KUKA KRL program: EPS_2_251455_MH62A_A_20251003045105.src

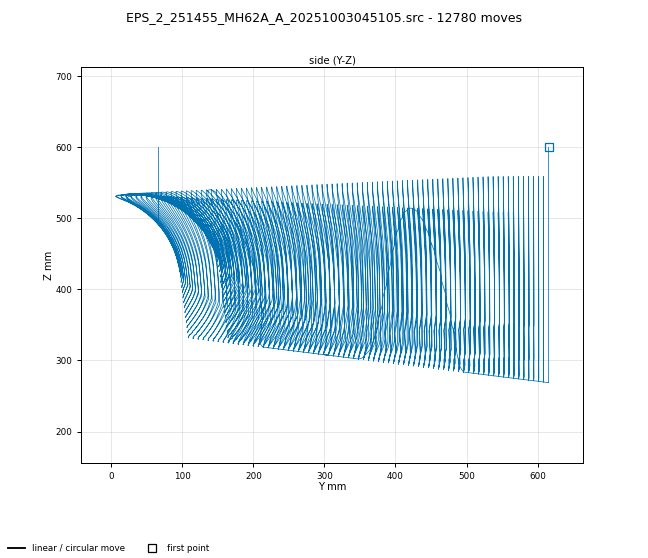
[picture p0: tool path of EPS_2_251455_MH62A_A_20251003045105.src, 12780 of 12782 moves have a stored position in this frame; points joined in program order, loops and branches not executed]
&ACCESS RVP
&REL 4
&COMMENT QRS 19112012
&PARAM EDITMASK = *
DEF PART()
EXT BAS (BAS_COMMAND :IN,REAL :IN )
INT I
BAS (#INITMOV,0 )

;KUKA QRS Post kuka4.cps  Date:22-06-2017 !

File_ID=2872

QRS_PRE_INIT()

;Init var - Until changes are made in qrs_pre_init
Outlet_Square_prg=0
Inlet_1_Square_prg=0
Inlet_2_Square_prg=0
Inlet_3_Square_prg=0
Inlet_4_Square_prg=0
Inlet_5_Square_prg=0

Outlet_1={X 0.000, Y 535.490, Z 458.500, B 0.000, E1 0.000 }
Inlet_1={X 0.000, Y 539.060, Z 408.500, B 0.000, E1 171.000 }
Outlet_1_type=201
Inlet_1_type=201
;QRS#1=Sidecore dimensions
;QRS#2=200-8" PVC SDR 35
;QRS#3=200-8" PVC SDR 35
;QRS#4=
;QRS#5=
;QRS#6=
;QRS#7=
;QRS#8=
;QRS#9=12-08 PSX
;QRS#10=12-08 PSX
;QRS#11=
;QRS#12=
;QRS#13=
;QRS#14=
;QRS#15=
;QRS#16=1220x127x838 2,75'
;QRS#17=EPS Height
;QRS#18=559
;QRS#19=*
;QRS#20= UPDATED VERSION 22-06-2017
;QRS#21=*
Outlet_Square=0100
Inlet_1_Square=0100
Inlet_2_Square=0
Inlet_3_Square=0
Inlet_4_Square=0
Inlet_5_Square=0
Mill_Square=1
Outlet_Square_Prg=204
Inlet_1_Square_prg=204

QRS_INIT()

$ADVANCE=5

; T1
PTP {E1 173.608,E2 173.608}
PTP {X 0,Y 615.498,A -85,B 0,C 180,E1 173.608,E2 173.608,E3 0,E4 0,E5 0,E6 0}
QRS_SPEED_INIT()
LIN {X 0,Y 615.498,Z 600,A -85,B 0,C 180,E1 173.608,E2 173.608,E3 0,E4 0,E5 0,E6 0} C_VEL
LIN {X 0,Y 615.498,Z 278.865,A -85,B 0,C 180,E1 173.608,E2 173.608} C_VEL
LIN {X 0,Y 615.498,Z 270.69,A -85,B 0,C 180,E1 173.608,E2 173.608} C_VEL
LIN {X 0,Y 615.483,Z 268.69,A -85,B 0,C 180,E1 173.422,E2 173.422} C_VEL
LIN {X 0,Y 615.481,Z 268.697,A -85,B 0,C 180,E1 170.801,E2 170.801} C_VEL
LIN {X 0,Y 615.465,Z 268.687,A -85,B 0,C 180,E1 168.139,E2 168.139} C_VEL
LIN {X 0,Y 615.488,Z 268.686,A -85,B 0,C 180,E1 165.451,E2 165.451} C_VEL
LIN {X 0,Y 615.481,Z 268.698,A -85,B 0,C 180,E1 162.729,E2 162.729} C_VEL
LIN {X 0,Y 615.462,Z 268.687,A -85,B 0,C 180,E1 159.966,E2 159.966} C_VEL
LIN {X 0,Y 615.49,Z 268.691,A -85,B 0,C 180,E1 157.155,E2 157.155} C_VEL
LIN {X 0,Y 615.457,Z 268.693,A -85,B 0,C 180,E1 154.283,E2 154.283} C_VEL
LIN {X 0,Y 615.452,Z 268.691,A -85,B 0,C 180,E1 152.083,E2 152.083} C_VEL
LIN {X 0,Y 615.455,Z 268.689,A -85,B 0,C 180,E1 149.838,E2 149.838} C_VEL
LIN {X 0,Y 615.47,Z 268.686,A -85,B 0,C 180,E1 147.541,E2 147.541} C_VEL
LIN {X 0,Y 615.498,Z 268.685,A -85,B 0,C 180,E1 145.185,E2 145.185} C_VEL
LIN {X 0,Y 615.491,Z 268.699,A -85,B 0,C 180,E1 142.758,E2 142.758} C_VEL
LIN {X 0,Y 615.454,Z 268.696,A -85,B 0,C 180,E1 140.247,E2 140.247} C_VEL
LIN {X 0,Y 615.441,Z 268.694,A -85,B 0,C 180,E1 137.924,E2 137.924} C_VEL
LIN {X 0,Y 615.436,Z 268.694,A -85,B 0,C 180,E1 135.845,E2 135.845} C_VEL
LIN {X 0,Y 615.46,Z 268.69,A -85,B 0,C 180,E1 133.246,E2 133.246} C_VEL
LIN {X 0,Y 615.493,Z 268.7,A -85,B 0,C 180,E1 130.605,E2 130.605} C_VEL
LIN {X 0,Y 615.438,Z 268.697,A -85,B 0,C 180,E1 128.005,E2 128.005} C_VEL
LIN {X 0,Y 615.429,Z 268.695,A -85,B 0,C 180,E1 125.619,E2 125.619} C_VEL
LIN {X 0,Y 615.44,Z 268.693,A -85,B 0,C 180,E1 123.239,E2 123.239} C_VEL
LIN {X 0,Y 615.464,Z 268.693,A -85,B 0,C 180,E1 120.921,E2 120.921} C_VEL
LIN {X 0,Y 615.436,Z 268.698,A -85,B 0,C 180,E1 117.917,E2 117.917} C_VEL
LIN {X 0,Y 615.449,Z 268.854,A -85,B 0,C 180,E1 116.961,E2 116.961} C_VEL
LIN {X 0,Y 615.469,Z 284.204,A -85,B 0,C 180,E1 114.272,E2 114.272} C_VEL
LIN {X 0,Y 615.472,Z 298.44,A -85,B 0,C 180,E1 111.806,E2 111.806} C_VEL
LIN {X 0,Y 615.492,Z 404.077,A -85,B 0,C 180,E1 110.557,E2 110.557} C_VEL
LIN {X 0,Y 615.488,Z 417.766,A -85,B 0,C 180,E1 110.262,E2 110.262} C_VEL
LIN {X 0,Y 615.49,Z 430.179,A -85,B 0,C 180,E1 109.858,E2 109.858} C_VEL
LIN {X 0,Y 615.47,Z 442.042,A -85,B 0,C 180,E1 109.338,E2 109.338} C_VEL
LIN {X 0,Y 615.471,Z 452.757,A -85,B 0,C 180,E1 108.732,E2 108.732} C_VEL
LIN {X 0,Y 615.499,Z 463.692,A -85,B 0,C 180,E1 107.956,E2 107.956} C_VEL
LIN {X 0,Y 615.497,Z 473.463,A -85,B 0,C 180,E1 107.099,E2 107.099} C_VEL
LIN {X 0,Y 615.497,Z 481.984,A -85,B 0,C 180,E1 106.168,E2 106.168} C_VEL
LIN {X 0,Y 615.497,Z 489.025,A -85,B 0,C 180,E1 105.225,E2 105.225} C_VEL
LIN {X 0,Y 615.497,Z 494.959,A -85,B 0,C 180,E1 104.241,E2 104.241} C_VEL
LIN {X 0,Y 615.496,Z 499.897,A -85,B 0,C 180,E1 103.201,E2 103.201} C_VEL
LIN {X 0,Y 615.497,Z 503.505,A -85,B 0,C 180,E1 102.195,E2 102.195} C_VEL
LIN {X 0,Y 615.495,Z 506.657,A -85,B 0,C 180,E1 100.889,E2 100.889} C_VEL
LIN {X 0,Y 615.497,Z 507.995,A -85,B 0,C 180,E1 99.862,E2 99.862} C_VEL
LIN {X 0,Y 615.496,Z 508.296,A -85,B 0,C 180,E1 98.536,E2 98.536} C_VEL
LIN {X 0,Y 615.496,Z 507.851,A -85,B 0,C 180,E1 97.875,E2 97.875} C_VEL
LIN {X 0,Y 615.496,Z 505.719,A -85,B 0,C 180,E1 96.556,E2 96.556} C_VEL
LIN {X 0,Y 615.498,Z 503.036,A -85,B 0,C 180,E1 95.569,E2 95.569} C_VEL
LIN {X 0,Y 615.495,Z 499.359,A -85,B 0,C 180,E1 94.584,E2 94.584} C_VEL
LIN {X 0,Y 615.495,Z 494.582,A -85,B 0,C 180,E1 93.6,E2 93.6} C_VEL
LIN {X 0,Y 615.497,Z 488.57,A -85,B 0,C 180,E1 92.617,E2 92.617} C_VEL
LIN {X 0,Y 615.498,Z 481.113,A -85,B 0,C 180,E1 91.635,E2 91.635} C_VEL
LIN {X 0,Y 615.498,Z 473.523,A -85,B 0,C 180,E1 90.817,E2 90.817} C_VEL
LIN {X 0,Y 615.498,Z 463.233,A -85,B 0,C 180,E1 89.918,E2 89.918} C_VEL
LIN {X 0,Y 615.467,Z 452.822,A -85,B 0,C 180,E1 89.182,E2 89.182} C_VEL
LIN {X 0,Y 615.466,Z 442.767,A -85,B 0,C 180,E1 88.609,E2 88.609} C_VEL
LIN {X 0,Y 615.496,Z 430.865,A -85,B 0,C 180,E1 88.077,E2 88.077} C_VEL
LIN {X 0,Y 615.47,Z 418.497,A -85,B 0,C 180,E1 87.668,E2 87.668} C_VEL
LIN {X 0,Y 615.455,Z 405.743,A -85,B 0,C 180,E1 87.382,E2 87.382} C_VEL
LIN {X 0,Y 615.499,Z 333.951,A -85,B 0,C 180,E1 86.522,E2 86.522} C_VEL
LIN {X 0,Y 615.492,Z 298.362,A -85,B 0,C 180,E1 86.092,E2 86.092} C_VEL
LIN {X 0,Y 615.49,Z 282.974,A -85,B 0,C 180,E1 83.425,E2 83.425} C_VEL
LIN {X 0,Y 615.439,Z 268.696,A -85,B 0,C 180,E1 80.904,E2 80.904} C_VEL
LIN {X 0,Y 615.434,Z 268.696,A -85,B 0,C 180,E1 78.806,E2 78.806} C_VEL
LIN {X 0,Y 615.438,Z 268.696,A -85,B 0,C 180,E1 76.797,E2 76.797} C_VEL
LIN {X 0,Y 615.438,Z 268.696,A -85,B 0,C 180,E1 74.772,E2 74.772} C_VEL
LIN {X 0,Y 615.435,Z 268.697,A -85,B 0,C 180,E1 72.728,E2 72.728} C_VEL
LIN {X 0,Y 615.436,Z 268.696,A -85,B 0,C 180,E1 70.66,E2 70.66} C_VEL
LIN {X 0,Y 615.435,Z 268.696,A -85,B 0,C 180,E1 68.566,E2 68.566} C_VEL
LIN {X 0,Y 615.433,Z 268.695,A -85,B 0,C 180,E1 66.441,E2 66.441} C_VEL
LIN {X 0,Y 615.429,Z 268.695,A -85,B 0,C 180,E1 64.281,E2 64.281} C_VEL
LIN {X 0,Y 615.433,Z 268.693,A -85,B 0,C 180,E1 62.082,E2 62.082} C_VEL
LIN {X 0,Y 615.491,Z 268.699,A -85,B 0,C 180,E1 59.08,E2 59.08} C_VEL
LIN {X 0,Y 615.444,Z 268.697,A -85,B 0,C 180,E1 56.473,E2 56.473} C_VEL
LIN {X 0,Y 615.432,Z 268.695,A -85,B 0,C 180,E1 54.174,E2 54.174} C_VEL
LIN {X 0,Y 615.431,Z 268.694,A -85,B 0,C 180,E1 51.927,E2 51.927} C_VEL
LIN {X 0,Y 615.459,Z 268.691,A -85,B 0,C 180,E1 49.391,E2 49.391} C_VEL
LIN {X 0,Y 615.498,Z 268.7,A -85,B 0,C 180,E1 46.756,E2 46.756} C_VEL
LIN {X 0,Y 615.44,Z 268.697,A -85,B 0,C 180,E1 44.154,E2 44.154} C_VEL
LIN {X 0,Y 615.439,Z 268.696,A -85,B 0,C 180,E1 42.075,E2 42.075} C_VEL
LIN {X 0,Y 615.43,Z 268.694,A -85,B 0,C 180,E1 39.755,E2 39.755} C_VEL
LIN {X 0,Y 615.448,Z 268.691,A -85,B 0,C 180,E1 37.245,E2 37.245} C_VEL
LIN {X 0,Y 615.493,Z 268.693,A -85,B 0,C 180,E1 34.701,E2 34.701} C_VEL
LIN {X 0,Y 615.487,Z 268.699,A -85,B 0,C 180,E1 32.33,E2 32.33} C_VEL
LIN {X 0,Y 615.437,Z 268.696,A -85,B 0,C 180,E1 29.786,E2 29.786} C_VEL
LIN {X 0,Y 615.449,Z 268.697,A -85,B 0,C 180,E1 27.917,E2 27.917} C_VEL
LIN {X 0,Y 615.432,Z 268.695,A -85,B 0,C 180,E1 25.557,E2 25.557} C_VEL
LIN {X 0,Y 615.433,Z 268.696,A -85,B 0,C 180,E1 23.559,E2 23.559} C_VEL
LIN {X 0,Y 615.431,Z 268.695,A -85,B 0,C 180,E1 21.434,E2 21.434} C_VEL
LIN {X 0,Y 615.429,Z 268.695,A -85,B 0,C 180,E1 19.34,E2 19.34} C_VEL
LIN {X 0,Y 615.428,Z 268.695,A -85,B 0,C 180,E1 17.273,E2 17.273} C_VEL
LIN {X 0,Y 615.43,Z 268.695,A -85,B 0,C 180,E1 15.228,E2 15.228} C_VEL
LIN {X 0,Y 615.43,Z 268.695,A -85,B 0,C 180,E1 13.203,E2 13.203} C_VEL
LIN {X 0,Y 615.434,Z 268.693,A -85,B 0,C 180,E1 10.86,E2 10.86} C_VEL
LIN {X 0,Y 615.454,Z 268.691,A -85,B 0,C 180,E1 8.537,E2 8.537} C_VEL
LIN {X 0,Y 615.498,Z 268.698,A -85,B 0,C 180,E1 5.899,E2 5.899} C_VEL
LIN {X 0,Y 615.441,Z 268.697,A -85,B 0,C 180,E1 3.273,E2 3.273} C_VEL
LIN {X 0,Y 615.447,Z 268.697,A -85,B 0,C 180,E1 1.309,E2 1.309} C_VEL
LIN {X 0,Y 615.454,Z 268.698,A -85,B 0,C 180,E1 -0.654,E2 -0.654} C_VEL
LIN {X 0,Y 615.462,Z 268.698,A -85,B 0,C 180,E1 -2.618,E2 -2.618} C_VEL
LIN {X 0,Y 615.428,Z 268.695,A -85,B 0,C 180,E1 -5.242,E2 -5.242} C_VEL
LIN {X 0,Y 615.429,Z 268.695,A -85,B 0,C 180,E1 -7.216,E2 -7.216} C_VEL
LIN {X 0,Y 615.431,Z 268.696,A -85,B 0,C 180,E1 -9.2,E2 -9.2} C_VEL
LIN {X 0,Y 615.431,Z 268.696,A -85,B 0,C 180,E1 -11.194,E2 -11.194} C_VEL
LIN {X 0,Y 615.434,Z 268.696,A -85,B 0,C 180,E1 -13.202,E2 -13.202} C_VEL
LIN {X 0,Y 615.435,Z 268.696,A -85,B 0,C 180,E1 -15.227,E2 -15.227} C_VEL
LIN {X 0,Y 615.435,Z 268.696,A -85,B 0,C 180,E1 -17.272,E2 -17.272} C_VEL
LIN {X 0,Y 615.432,Z 268.696,A -85,B 0,C 180,E1 -19.34,E2 -19.34} C_VEL
LIN {X 0,Y 615.432,Z 268.696,A -85,B 0,C 180,E1 -21.434,E2 -21.434} C_VEL
LIN {X 0,Y 615.429,Z 268.695,A -85,B 0,C 180,E1 -23.559,E2 -23.559} C_VEL
LIN {X 0,Y 615.428,Z 268.695,A -85,B 0,C 180,E1 -25.718,E2 -25.718} C_VEL
LIN {X 0,Y 615.43,Z 268.694,A -85,B 0,C 180,E1 -27.918,E2 -27.918} C_VEL
LIN {X 0,Y 615.491,Z 268.7,A -85,B 0,C 180,E1 -30.92,E2 -30.92} C_VEL
LIN {X 0,Y 615.438,Z 268.698,A -85,B 0,C 180,E1 -33.526,E2 -33.526} C_VEL
LIN {X 0,Y 615.429,Z 268.695,A -85,B 0,C 180,E1 -35.825,E2 -35.825} C_VEL
LIN {X 0,Y 615.428,Z 268.694,A -85,B 0,C 180,E1 -38.073,E2 -38.073} C_VEL
LIN {X 0,Y 615.427,Z 268.695,A -85,B 0,C 180,E1 -40.082,E2 -40.082} C_VEL
LIN {X 0,Y 615.435,Z 268.693,A -85,B 0,C 180,E1 -42.358,E2 -42.358} C_VEL
LIN {X 0,Y 615.497,Z 268.693,A -85,B 0,C 180,E1 -45.068,E2 -45.068} C_VEL
LIN {X 0,Y 615.435,Z 268.697,A -85,B 0,C 180,E1 -47.925,E2 -47.925} C_VEL
LIN {X 0,Y 615.427,Z 268.695,A -85,B 0,C 180,E1 -50.245,E2 -50.245} C_VEL
LIN {X 0,Y 615.447,Z 268.692,A -85,B 0,C 180,E1 -52.754,E2 -52.754} C_VEL
LIN {X 0,Y 615.496,Z 268.693,A -85,B 0,C 180,E1 -55.299,E2 -55.299} C_VEL
LIN {X 0,Y 615.481,Z 268.699,A -85,B 0,C 180,E1 -57.671,E2 -57.671} C_VEL
LIN {X 0,Y 615.433,Z 268.696,A -85,B 0,C 180,E1 -60.215,E2 -60.215} C_VEL
LIN {X 0,Y 615.445,Z 268.697,A -85,B 0,C 180,E1 -62.082,E2 -62.082} C_VEL
LIN {X 0,Y 615.428,Z 268.696,A -85,B 0,C 180,E1 -64.443,E2 -64.443} C_VEL
LIN {X 0,Y 615.43,Z 268.694,A -85,B 0,C 180,E1 -66.797,E2 -66.797} C_VEL
LIN {X 0,Y 615.446,Z 268.819,A -85,B 0,C 180,E1 -67.065,E2 -67.065} C_VEL
LIN {X 0,Y 615.472,Z 290.751,A -85,B 0,C 180,E1 -69.966,E2 -69.966} C_VEL
LIN {X 0,Y 615.457,Z 310.668,A -85,B 0,C 180,E1 -72.557,E2 -72.557} C_VEL
LIN {X 0,Y 615.484,Z 331.887,A -85,B 0,C 180,E1 -75.281,E2 -75.281} C_VEL
LIN {X 0,Y 615.459,Z 346.297,A -85,B 0,C 180,E1 -77.113,E2 -77.113} C_VEL
LIN {X 0,Y 615.454,Z 454.814,A -85,B 0,C 180,E1 -78.41,E2 -78.41} C_VEL
LIN {X 0,Y 615.454,Z 467.335,A -85,B 0,C 180,E1 -78.681,E2 -78.681} C_VEL
LIN {X 0,Y 615.482,Z 480.695,A -85,B 0,C 180,E1 -79.116,E2 -79.116} C_VEL
LIN {X 0,Y 615.492,Z 492.468,A -85,B 0,C 180,E1 -79.639,E2 -79.639} C_VEL
LIN {X 0,Y 615.486,Z 503.989,A -85,B 0,C 180,E1 -80.303,E2 -80.303} C_VEL
LIN {X 0,Y 615.499,Z 514.336,A -85,B 0,C 180,E1 -81.049,E2 -81.049} C_VEL
LIN {X 0,Y 615.497,Z 522.807,A -85,B 0,C 180,E1 -81.794,E2 -81.794} C_VEL
LIN {X 0,Y 615.498,Z 530.603,A -85,B 0,C 180,E1 -82.619,E2 -82.619} C_VEL
LIN {X 0,Y 615.497,Z 538.2,A -85,B 0,C 180,E1 -83.608,E2 -83.608} C_VEL
LIN {X 0,Y 615.498,Z 545.202,A -85,B 0,C 180,E1 -84.758,E2 -84.758} C_VEL
LIN {X 0,Y 615.494,Z 549.849,A -85,B 0,C 180,E1 -85.743,E2 -85.743} C_VEL
LIN {X 0,Y 615.494,Z 553.397,A -85,B 0,C 180,E1 -86.727,E2 -86.727} C_VEL
LIN {X 0,Y 615.497,Z 555.232,A -85,B 0,C 180,E1 -87.382,E2 -87.382} C_VEL
LIN {X 0,Y 615.498,Z 556.607,A -85,B 0,C 180,E1 -88.037,E2 -88.037} C_VEL
LIN {X 0,Y 615.496,Z 558.173,A -85,B 0,C 180,E1 -89.345,E2 -89.345} C_VEL
LIN {X 0,Y 615.494,Z 558.389,A -85,B 0,C 180,E1 -90,E2 -90} C_VEL
LIN {X 0,Y 615.495,Z 557.581,A -85,B 0,C 180,E1 -91.308,E2 -91.308} C_VEL
LIN {X 0,Y 615.498,Z 556.609,A -85,B 0,C 180,E1 -91.963,E2 -91.963} C_VEL
LIN {X 0,Y 615.497,Z 555.234,A -85,B 0,C 180,E1 -92.617,E2 -92.617} C_VEL
LIN {X 0,Y 615.496,Z 552.351,A -85,B 0,C 180,E1 -93.6,E2 -93.6} C_VEL
LIN {X 0,Y 615.498,Z 548.443,A -85,B 0,C 180,E1 -94.584,E2 -94.584} C_VEL
LIN {X 0,Y 615.499,Z 543.407,A -85,B 0,C 180,E1 -95.569,E2 -95.569} C_VEL
LIN {X 0,Y 615.497,Z 536.869,A -85,B 0,C 180,E1 -96.583,E2 -96.583} C_VEL
LIN {X 0,Y 615.497,Z 529.137,A -85,B 0,C 180,E1 -97.545,E2 -97.545} C_VEL
LIN {X 0,Y 615.498,Z 521.049,A -85,B 0,C 180,E1 -98.371,E2 -98.371} C_VEL
LIN {X 0,Y 615.499,Z 511.173,A -85,B 0,C 180,E1 -99.198,E2 -99.198} C_VEL
LIN {X 0,Y 615.486,Z 499.989,A -85,B 0,C 180,E1 -99.945,E2 -99.945} C_VEL
LIN {X 0,Y 615.493,Z 489.03,A -85,B 0,C 180,E1 -100.526,E2 -100.526} C_VEL
LIN {X 0,Y 615.468,Z 476.539,A -85,B 0,C 180,E1 -101.039,E2 -101.039} C_VEL
LIN {X 0,Y 615.452,Z 464.091,A -85,B 0,C 180,E1 -101.402,E2 -101.402} C_VEL
LIN {X 0,Y 615.456,Z 450.505,A -85,B 0,C 180,E1 -101.652,E2 -101.652} C_VEL
LIN {X 0,Y 615.459,Z 346.303,A -85,B 0,C 180,E1 -102.887,E2 -102.887} C_VEL
LIN {X 0,Y 615.468,Z 326.591,A -85,B 0,C 180,E1 -105.396,E2 -105.396} C_VEL
LIN {X 0,Y 615.493,Z 304.197,A -85,B 0,C 180,E1 -108.28,E2 -108.28} C_VEL
LIN {X 0,Y 615.469,Z 282.785,A -85,B 0,C 180,E1 -111.081,E2 -111.081} C_VEL
LIN {X 0,Y 615.444,Z 268.693,A -85,B 0,C 180,E1 -112.979,E2 -112.979} C_VEL
LIN {X 0,Y 615.447,Z 268.692,A -85,B 0,C 180,E1 -114.993,E2 -114.993} C_VEL
LIN {X 0,Y 615.439,Z 268.693,A -85,B 0,C 180,E1 -117.179,E2 -117.179} C_VEL
LIN {X 0,Y 615.435,Z 268.693,A -85,B 0,C 180,E1 -119.409,E2 -119.409} C_VEL
LIN {X 0,Y 615.439,Z 268.695,A -85,B 0,C 180,E1 -121.688,E2 -121.688} C_VEL
LIN {X 0,Y 615.46,Z 268.697,A -85,B 0,C 180,E1 -124.023,E2 -124.023} C_VEL
LIN {X 0,Y 615.476,Z 268.688,A -85,B 0,C 180,E1 -126.935,E2 -126.935} C_VEL
LIN {X 0,Y 615.445,Z 268.694,A -85,B 0,C 180,E1 -129.753,E2 -129.753} C_VEL
LIN {X 0,Y 615.488,Z 268.699,A -85,B 0,C 180,E1 -132.352,E2 -132.352} C_VEL
LIN {X 0,Y 615.492,Z 268.684,A -85,B 0,C 180,E1 -135.068,E2 -135.068} C_VEL
LIN {X 0,Y 615.452,Z 268.69,A -85,B 0,C 180,E1 -137.644,E2 -137.644} C_VEL
LIN {X 0,Y 615.471,Z 268.697,A -85,B 0,C 180,E1 -140.248,E2 -140.248} C_VEL
LIN {X 0,Y 615.486,Z 268.687,A -85,B 0,C 180,E1 -143.063,E2 -143.063} C_VEL
LIN {X 0,Y 615.486,Z 268.683,A -85,B 0,C 180,E1 -145.299,E2 -145.299} C_VEL
LIN {X 0,Y 615.466,Z 268.686,A -85,B 0,C 180,E1 -147.672,E2 -147.672} C_VEL
LIN {X 0,Y 615.466,Z 268.694,A -85,B 0,C 180,E1 -150.208,E2 -150.208} C_VEL
LIN {X 0,Y 615.482,Z 268.693,A -85,B 0,C 180,E1 -152.955,E2 -152.955} C_VEL
LIN {X 0,Y 615.476,Z 268.684,A -85,B 0,C 180,E1 -155.728,E2 -155.728} C_VEL
LIN {X 0,Y 615.485,Z 268.698,A -85,B 0,C 180,E1 -158.568,E2 -158.568} C_VEL
LIN {X 0,Y 615.488,Z 268.684,A -85,B 0,C 180,E1 -161.394,E2 -161.394} C_VEL
LIN {X 0,Y 615.471,Z 268.687,A -85,B 0,C 180,E1 -164.094,E2 -164.094} C_VEL
LIN {X 0,Y 615.496,Z 268.701,A -85,B 0,C 180,E1 -166.799,E2 -166.799} C_VEL
LIN {X 0,Y 615.482,Z 268.685,A -85,B 0,C 180,E1 -169.473,E2 -169.473} C_VEL
LIN {X 0,Y 615.479,Z 268.685,A -85,B 0,C 180,E1 -172.124,E2 -172.124} C_VEL
LIN {X 0,Y 615.487,Z 268.699,A -85,B 0,C 180,E1 -174.759,E2 -174.759} C_VEL
LIN {X 0,Y 615.474,Z 268.69,A -85,B 0,C 180,E1 -177.382,E2 -177.382} C_VEL
LIN {X 0,Y 615.486,Z 268.682,A -85,B 0,C 180,E1 -180,E2 -180} C_VEL
LIN {X 0,Y 615.482,Z 268.692,A -85,B 0,C 180,E1 -182.618,E2 -182.618} C_VEL
LIN {X 0,Y 615.478,Z 268.695,A -85,B 0,C 180,E1 -185.241,E2 -185.241} C_VEL
LIN {X 0,Y 615.483,Z 268.69,A -85,B 0,C 180,E1 -186.578,E2 -186.578} C_VEL
LIN {X 0,Y 614.806,Z 268.843,A -85,B 0,C 180,E1 -187.124,E2 -187.124} C_VEL
LIN {X 0,Y 611.972,Z 269.248,A -85,B 0,C 180,E1 -188.01,E2 -188.01} C_VEL
LIN {X 0,Y 609.58,Z 269.563,A -85,B 0,C 180,E1 -188.722,E2 -188.722} C_VEL
LIN {X 0,Y 608.543,Z 269.682,A -85,B 0,C 180,E1 -189.272,E2 -189.272} C_VEL
LIN {X 0,Y 608.452,Z 269.691,A -85,B 0,C 180,E1 -189.458,E2 -189.458} C_VEL
LIN {X 0,Y 608.447,Z 269.687,A -85,B 0,C 180,E1 -192,E2 -192} C_VEL
LIN {X 0,Y 608.476,Z 269.689,A -85,B 0,C 180,E1 -194.721,E2 -194.721} C_VEL
LIN {X 0,Y 608.443,Z 269.693,A -85,B 0,C 180,E1 -197.477,E2 -197.477} C_VEL
LIN {X 0,Y 608.439,Z 269.692,A -85,B 0,C 180,E1 -199.571,E2 -199.571} C_VEL
LIN {X 0,Y 608.475,Z 269.685,A -85,B 0,C 180,E1 -202.406,E2 -202.406} C_VEL
LIN {X 0,Y 608.441,Z 269.697,A -85,B 0,C 180,E1 -205.302,E2 -205.302} C_VEL
LIN {X 0,Y 608.436,Z 269.694,A -85,B 0,C 180,E1 -207.519,E2 -207.519} C_VEL
LIN {X 0,Y 608.438,Z 269.689,A -85,B 0,C 180,E1 -209.968,E2 -209.968} C_VEL
LIN {X 0,Y 608.453,Z 269.691,A -85,B 0,C 180,E1 -212.88,E2 -212.88} C_VEL
LIN {X 0,Y 608.436,Z 269.7,A -85,B 0,C 180,E1 -215.279,E2 -215.279} C_VEL
LIN {X 0,Y 608.445,Z 269.691,A -85,B 0,C 180,E1 -217.748,E2 -217.748} C_VEL
LIN {X 0,Y 608.432,Z 269.689,A -85,B 0,C 180,E1 -220.327,E2 -220.327} C_VEL
LIN {X 0,Y 608.455,Z 269.691,A -85,B 0,C 180,E1 -222.96,E2 -222.96} C_VEL
LIN {X 0,Y 608.426,Z 269.695,A -85,B 0,C 180,E1 -225.74,E2 -225.74} C_VEL
LIN {X 0,Y 608.428,Z 269.693,A -85,B 0,C 180,E1 -227.936,E2 -227.936} C_VEL
LIN {X 0,Y 608.425,Z 269.691,A -85,B 0,C 180,E1 -230.708,E2 -230.708} C_VEL
LIN {X 0,Y 608.445,Z 269.692,A -85,B 0,C 180,E1 -233.085,E2 -233.085} C_VEL
LIN {X 0,Y 608.464,Z 269.696,A -85,B 0,C 180,E1 -235.531,E2 -235.531} C_VEL
LIN {X 0,Y 608.442,Z 269.693,A -85,B 0,C 180,E1 -237.905,E2 -237.905} C_VEL
LIN {X 0,Y 608.416,Z 269.693,A -85,B 0,C 180,E1 -240.218,E2 -240.218} C_VEL
LIN {X 0,Y 608.408,Z 269.693,A -85,B 0,C 180,E1 -242.48,E2 -242.48} C_VEL
LIN {X 0,Y 608.435,Z 269.725,A -85,B 0,C 180,E1 -242.964,E2 -242.964} C_VEL
LIN {X 0,Y 608.455,Z 286.087,A -85,B 0,C 180,E1 -245.854,E2 -245.854} C_VEL
LIN {X 0,Y 608.451,Z 298.63,A -85,B 0,C 180,E1 -248.041,E2 -248.041} C_VEL
LIN {X 0,Y 608.541,Z 405.447,A -85,B 0,C 180,E1 -249.331,E2 -249.331} C_VEL
LIN {X 0,Y 608.536,Z 419.262,A -85,B 0,C 180,E1 -249.646,E2 -249.646} C_VEL
LIN {X 0,Y 608.518,Z 432.022,A -85,B 0,C 180,E1 -250.081,E2 -250.081} C_VEL
LIN {X 0,Y 608.483,Z 443.433,A -85,B 0,C 180,E1 -250.606,E2 -250.606} C_VEL
LIN {X 0,Y 608.469,Z 454.966,A -85,B 0,C 180,E1 -251.286,E2 -251.286} C_VEL
LIN {X 0,Y 608.478,Z 465.839,A -85,B 0,C 180,E1 -252.09,E2 -252.09} C_VEL
LIN {X 0,Y 608.462,Z 476.082,A -85,B 0,C 180,E1 -253.044,E2 -253.044} C_VEL
LIN {X 0,Y 608.462,Z 484.996,A -85,B 0,C 180,E1 -254.079,E2 -254.079} C_VEL
LIN {X 0,Y 608.451,Z 492.05,A -85,B 0,C 180,E1 -255.108,E2 -255.108} C_VEL
LIN {X 0,Y 608.432,Z 498.55,A -85,B 0,C 180,E1 -256.319,E2 -256.319} C_VEL
LIN {X 0,Y 608.427,Z 502.613,A -85,B 0,C 180,E1 -257.322,E2 -257.322} C_VEL
LIN {X 0,Y 608.444,Z 504.752,A -85,B 0,C 180,E1 -258,E2 -258} C_VEL
LIN {X 0,Y 608.423,Z 507.219,A -85,B 0,C 180,E1 -259.07,E2 -259.07} C_VEL
LIN {X 0,Y 608.433,Z 508.527,A -85,B 0,C 180,E1 -260.023,E2 -260.023} C_VEL
LIN {X 0,Y 608.419,Z 508.931,A -85,B 0,C 180,E1 -261.364,E2 -261.364} C_VEL
LIN {X 0,Y 608.42,Z 508.554,A -85,B 0,C 180,E1 -262.033,E2 -262.033} C_VEL
LIN {X 0,Y 608.42,Z 507.75,A -85,B 0,C 180,E1 -262.7,E2 -262.7} C_VEL
LIN {X 0,Y 608.448,Z 506.462,A -85,B 0,C 180,E1 -263.398,E2 -263.398} C_VEL
LIN {X 0,Y 608.441,Z 502.859,A -85,B 0,C 180,E1 -264.698,E2 -264.698} C_VEL
LIN {X 0,Y 608.442,Z 498.899,A -85,B 0,C 180,E1 -265.695,E2 -265.695} C_VEL
LIN {X 0,Y 608.457,Z 492.818,A -85,B 0,C 180,E1 -266.855,E2 -266.855} C_VEL
LIN {X 0,Y 608.453,Z 486.2,A -85,B 0,C 180,E1 -267.849,E2 -267.849} C_VEL
LIN {X 0,Y 608.479,Z 478.013,A -85,B 0,C 180,E1 -268.842,E2 -268.842} C_VEL
LIN {X 0,Y 608.469,Z 469.665,A -85,B 0,C 180,E1 -269.67,E2 -269.67} C_VEL
LIN {X 0,Y 608.479,Z 459.39,A -85,B 0,C 180,E1 -270.497,E2 -270.497} C_VEL
LIN {X 0,Y 608.455,Z 447.897,A -85,B 0,C 180,E1 -271.241,E2 -271.241} C_VEL
LIN {X 0,Y 608.502,Z 436.461,A -85,B 0,C 180,E1 -271.821,E2 -271.821} C_VEL
LIN {X 0,Y 608.509,Z 423.446,A -85,B 0,C 180,E1 -272.317,E2 -272.317} C_VEL
LIN {X 0,Y 608.501,Z 410.286,A -85,B 0,C 180,E1 -272.669,E2 -272.669} C_VEL
LIN {X 0,Y 608.504,Z 395.451,A -85,B 0,C 180,E1 -272.897,E2 -272.897} C_VEL
LIN {X 0,Y 608.539,Z 299.156,A -85,B 0,C 180,E1 -274.036,E2 -274.036} C_VEL
LIN {X 0,Y 608.46,Z 298.582,A -85,B 0,C 180,E1 -274.057,E2 -274.057} C_VEL
LIN {X 0,Y 608.481,Z 281.927,A -85,B 0,C 180,E1 -276.966,E2 -276.966} C_VEL
LIN {X 0,Y 608.434,Z 269.691,A -85,B 0,C 180,E1 -279.139,E2 -279.139} C_VEL
LIN {X 0,Y 608.414,Z 269.692,A -85,B 0,C 180,E1 -281.325,E2 -281.325} C_VEL
LIN {X 0,Y 608.421,Z 269.691,A -85,B 0,C 180,E1 -283.358,E2 -283.358} C_VEL
LIN {X 0,Y 608.43,Z 269.69,A -85,B 0,C 180,E1 -285.407,E2 -285.407} C_VEL
LIN {X 0,Y 608.41,Z 269.692,A -85,B 0,C 180,E1 -287.478,E2 -287.478} C_VEL
LIN {X 0,Y 608.411,Z 269.692,A -85,B 0,C 180,E1 -289.572,E2 -289.572} C_VEL
LIN {X 0,Y 608.429,Z 269.689,A -85,B 0,C 180,E1 -291.693,E2 -291.693} C_VEL
LIN {X 0,Y 608.441,Z 269.694,A -85,B 0,C 180,E1 -294.572,E2 -294.572} C_VEL
LIN {X 0,Y 608.421,Z 269.692,A -85,B 0,C 180,E1 -297.52,E2 -297.52} C_VEL
LIN {X 0,Y 608.405,Z 269.692,A -85,B 0,C 180,E1 -299.96,E2 -299.96} C_VEL
LIN {X 0,Y 608.444,Z 269.69,A -85,B 0,C 180,E1 -302.519,E2 -302.519} C_VEL
LIN {X 0,Y 608.425,Z 269.698,A -85,B 0,C 180,E1 -305.279,E2 -305.279} C_VEL
LIN {X 0,Y 608.435,Z 269.69,A -85,B 0,C 180,E1 -307.749,E2 -307.749} C_VEL
LIN {X 0,Y 608.409,Z 269.692,A -85,B 0,C 180,E1 -310.323,E2 -310.323} C_VEL
LIN {X 0,Y 608.455,Z 269.692,A -85,B 0,C 180,E1 -312.96,E2 -312.96} C_VEL
LIN {X 0,Y 608.42,Z 269.695,A -85,B 0,C 180,E1 -315.74,E2 -315.74} C_VEL
LIN {X 0,Y 608.423,Z 269.692,A -85,B 0,C 180,E1 -317.935,E2 -317.935} C_VEL
LIN {X 0,Y 608.426,Z 269.691,A -85,B 0,C 180,E1 -320.708,E2 -320.708} C_VEL
LIN {X 0,Y 608.445,Z 269.692,A -85,B 0,C 180,E1 -323.084,E2 -323.084} C_VEL
LIN {X 0,Y 608.464,Z 269.697,A -85,B 0,C 180,E1 -325.53,E2 -325.53} C_VEL
LIN {X 0,Y 608.451,Z 269.692,A -85,B 0,C 180,E1 -327.904,E2 -327.904} C_VEL
LIN {X 0,Y 608.426,Z 269.692,A -85,B 0,C 180,E1 -330.218,E2 -330.218} C_VEL
LIN {X 0,Y 608.416,Z 269.691,A -85,B 0,C 180,E1 -332.48,E2 -332.48} C_VEL
LIN {X 0,Y 608.441,Z 269.693,A -85,B 0,C 180,E1 -335.428,E2 -335.428} C_VEL
LIN {X 0,Y 608.438,Z 269.691,A -85,B 0,C 180,E1 -338.307,E2 -338.307} C_VEL
LIN {X 0,Y 608.418,Z 269.693,A -85,B 0,C 180,E1 -340.428,E2 -340.428} C_VEL
LIN {X 0,Y 608.424,Z 269.691,A -85,B 0,C 180,E1 -343.215,E2 -343.215} C_VEL
LIN {X 0,Y 608.48,Z 269.695,A -85,B 0,C 180,E1 -345.981,E2 -345.981} C_VEL
LIN {X 0,Y 608.415,Z 269.693,A -85,B 0,C 180,E1 -348.675,E2 -348.675} C_VEL
LIN {X 0,Y 608.429,Z 269.691,A -85,B 0,C 180,E1 -350.693,E2 -350.693} C_VEL
LIN {X 0,Y 608.416,Z 269.693,A -85,B 0,C 180,E1 -352.7,E2 -352.7} C_VEL
LIN {X 0,Y 608.424,Z 269.693,A -85,B 0,C 180,E1 -354.698,E2 -354.698} C_VEL
LIN {X 0,Y 608.433,Z 269.689,A -85,B 0,C 180,E1 -357.352,E2 -357.352} C_VEL
LIN {X 0,Y 608.477,Z 269.689,A -85,B 0,C 180,E1 -360,E2 -360} C_VEL
LIN {X 0,Y 608.454,Z 269.692,A -85,B 0,C 180,E1 -362.648,E2 -362.648} C_VEL
LIN {X 0,Y 608.414,Z 269.691,A -85,B 0,C 180,E1 -365.302,E2 -365.302} C_VEL
LIN {X 0,Y 608.411,Z 269.692,A -85,B 0,C 180,E1 -367.3,E2 -367.3} C_VEL
LIN {X 0,Y 608.432,Z 269.692,A -85,B 0,C 180,E1 -369.978,E2 -369.978} C_VEL
LIN {X 0,Y 608.469,Z 269.694,A -85,B 0,C 180,E1 -372.677,E2 -372.677} C_VEL
LIN {X 0,Y 608.427,Z 269.69,A -85,B 0,C 180,E1 -375.407,E2 -375.407} C_VEL
LIN {X 0,Y 608.41,Z 269.692,A -85,B 0,C 180,E1 -377.478,E2 -377.478} C_VEL
LIN {X 0,Y 608.408,Z 269.692,A -85,B 0,C 180,E1 -379.572,E2 -379.572} C_VEL
LIN {X 0,Y 608.427,Z 269.69,A -85,B 0,C 180,E1 -381.693,E2 -381.693} C_VEL
LIN {X 0,Y 608.439,Z 269.695,A -85,B 0,C 180,E1 -384.572,E2 -384.572} C_VEL
LIN {X 0,Y 608.418,Z 269.692,A -85,B 0,C 180,E1 -387.52,E2 -387.52} C_VEL
LIN {X 0,Y 608.402,Z 269.693,A -85,B 0,C 180,E1 -389.96,E2 -389.96} C_VEL
LIN {X 0,Y 608.443,Z 269.691,A -85,B 0,C 180,E1 -392.519,E2 -392.519} C_VEL
LIN {X 0,Y 608.422,Z 269.698,A -85,B 0,C 180,E1 -395.279,E2 -395.279} C_VEL
LIN {X 0,Y 608.432,Z 269.691,A -85,B 0,C 180,E1 -397.749,E2 -397.749} C_VEL
LIN {X 0,Y 608.406,Z 269.692,A -85,B 0,C 180,E1 -400.323,E2 -400.323} C_VEL
LIN {X 0,Y 608.455,Z 269.693,A -85,B 0,C 180,E1 -402.96,E2 -402.96} C_VEL
LIN {X 0,Y 608.417,Z 269.695,A -85,B 0,C 180,E1 -405.74,E2 -405.74} C_VEL
LIN {X 0,Y 608.419,Z 269.693,A -85,B 0,C 180,E1 -407.935,E2 -407.935} C_VEL
LIN {X 0,Y 608.424,Z 269.691,A -85,B 0,C 180,E1 -410.708,E2 -410.708} C_VEL
LIN {X 0,Y 608.445,Z 269.692,A -85,B 0,C 180,E1 -413.084,E2 -413.084} C_VEL
LIN {X 0,Y 608.464,Z 269.696,A -85,B 0,C 180,E1 -415.53,E2 -415.53} C_VEL
LIN {X 0,Y 608.446,Z 269.692,A -85,B 0,C 180,E1 -417.904,E2 -417.904} C_VEL
LIN {X 0,Y 608.422,Z 269.692,A -85,B 0,C 180,E1 -420.218,E2 -420.218} C_VEL
LIN {X 0,Y 608.413,Z 269.692,A -85,B 0,C 180,E1 -422.48,E2 -422.48} C_VEL
LIN {X 0,Y 608.439,Z 269.694,A -85,B 0,C 180,E1 -425.428,E2 -425.428} C_VEL
LIN {X 0,Y 608.438,Z 269.817,A -85,B 0,C 180,E1 -426.92,E2 -426.92} C_VEL
LIN {X 0,Y 608.538,Z 282.78,A -85,B 0,C 180,E1 -428.666,E2 -428.666} C_VEL
LIN {X 0,Y 608.522,Z 302.448,A -85,B 0,C 180,E1 -431.271,E2 -431.271} C_VEL
LIN {X 0,Y 608.473,Z 323.998,A -85,B 0,C 180,E1 -434.078,E2 -434.078} C_VEL
LIN {X 0,Y 608.461,Z 343.942,A -85,B 0,C 180,E1 -436.643,E2 -436.643} C_VEL
LIN {X 0,Y 608.455,Z 346.518,A -85,B 0,C 180,E1 -436.972,E2 -436.972} C_VEL
LIN {X 0,Y 608.519,Z 454.924,A -85,B 0,C 180,E1 -438.276,E2 -438.276} C_VEL
LIN {X 0,Y 608.489,Z 468.201,A -85,B 0,C 180,E1 -438.571,E2 -438.571} C_VEL
LIN {X 0,Y 608.511,Z 480.65,A -85,B 0,C 180,E1 -438.983,E2 -438.983} C_VEL
LIN {X 0,Y 608.512,Z 492.627,A -85,B 0,C 180,E1 -439.519,E2 -439.519} C_VEL
LIN {X 0,Y 608.475,Z 504.191,A -85,B 0,C 180,E1 -440.191,E2 -440.191} C_VEL
LIN {X 0,Y 608.485,Z 514.588,A -85,B 0,C 180,E1 -440.945,E2 -440.945} C_VEL
LIN {X 0,Y 608.475,Z 523.107,A -85,B 0,C 180,E1 -441.698,E2 -441.698} C_VEL
LIN {X 0,Y 608.471,Z 530.957,A -85,B 0,C 180,E1 -442.533,E2 -442.533} C_VEL
LIN {X 0,Y 608.461,Z 538.283,A -85,B 0,C 180,E1 -443.484,E2 -443.484} C_VEL
LIN {X 0,Y 608.45,Z 543.864,A -85,B 0,C 180,E1 -444.365,E2 -444.365} C_VEL
LIN {X 0,Y 608.432,Z 548.948,A -85,B 0,C 180,E1 -445.362,E2 -445.362} C_VEL
LIN {X 0,Y 608.449,Z 552.895,A -85,B 0,C 180,E1 -446.357,E2 -446.357} C_VEL
LIN {X 0,Y 608.425,Z 555.808,A -85,B 0,C 180,E1 -447.351,E2 -447.351} C_VEL
LIN {X 0,Y 608.443,Z 557.201,A -85,B 0,C 180,E1 -448.014,E2 -448.014} C_VEL
LIN {X 0,Y 608.438,Z 558.783,A -85,B 0,C 180,E1 -449.338,E2 -449.338} C_VEL
LIN {X 0,Y 608.434,Z 559,A -85,B 0,C 180,E1 -450,E2 -450} C_VEL
LIN {X 0,Y 608.448,Z 558.184,A -85,B 0,C 180,E1 -451.323,E2 -451.323} C_VEL
LIN {X 0,Y 608.443,Z 557.202,A -85,B 0,C 180,E1 -451.985,E2 -451.985} C_VEL
LIN {X 0,Y 608.425,Z 555.81,A -85,B 0,C 180,E1 -452.648,E2 -452.648} C_VEL
LIN {X 0,Y 608.449,Z 552.898,A -85,B 0,C 180,E1 -453.642,E2 -453.642} C_VEL
LIN {X 0,Y 608.432,Z 548.952,A -85,B 0,C 180,E1 -454.637,E2 -454.637} C_VEL
LIN {X 0,Y 608.437,Z 542.879,A -85,B 0,C 180,E1 -455.8,E2 -455.8} C_VEL
LIN {X 0,Y 608.462,Z 536.238,A -85,B 0,C 180,E1 -456.799,E2 -456.799} C_VEL
LIN {X 0,Y 608.455,Z 527.993,A -85,B 0,C 180,E1 -457.8,E2 -457.8} C_VEL
LIN {X 0,Y 608.472,Z 519.541,A -85,B 0,C 180,E1 -458.635,E2 -458.635} C_VEL
LIN {X 0,Y 608.476,Z 509.097,A -85,B 0,C 180,E1 -459.473,E2 -459.473} C_VEL
LIN {X 0,Y 608.485,Z 498.763,A -85,B 0,C 180,E1 -460.144,E2 -460.144} C_VEL
LIN {X 0,Y 608.517,Z 487.611,A -85,B 0,C 180,E1 -460.724,E2 -460.724} C_VEL
LIN {X 0,Y 608.511,Z 475.915,A -85,B 0,C 180,E1 -461.192,E2 -461.192} C_VEL
LIN {X 0,Y 608.518,Z 463.285,A -85,B 0,C 180,E1 -461.555,E2 -461.555} C_VEL
LIN {X 0,Y 608.519,Z 450.632,A -85,B 0,C 180,E1 -461.787,E2 -461.787} C_VEL
LIN {X 0,Y 608.443,Z 346.442,A -85,B 0,C 180,E1 -463.038,E2 -463.038} C_VEL
LIN {X 0,Y 608.498,Z 327.994,A -85,B 0,C 180,E1 -465.405,E2 -465.405} C_VEL
LIN {X 0,Y 608.543,Z 305.471,A -85,B 0,C 180,E1 -468.332,E2 -468.332} C_VEL
LIN {X 0,Y 608.546,Z 284.117,A -85,B 0,C 180,E1 -471.155,E2 -471.155} C_VEL
LIN {X 0,Y 608.493,Z 270.156,A -85,B 0,C 180,E1 -473.032,E2 -473.032} C_VEL
LIN {X 0,Y 608.415,Z 269.694,A -85,B 0,C 180,E1 -473.125,E2 -473.125} C_VEL
LIN {X 0,Y 608.432,Z 269.692,A -85,B 0,C 180,E1 -475.713,E2 -475.713} C_VEL
LIN {X 0,Y 608.476,Z 269.689,A -85,B 0,C 180,E1 -478.62,E2 -478.62} C_VEL
LIN {X 0,Y 608.43,Z 269.69,A -85,B 0,C 180,E1 -481.318,E2 -481.318} C_VEL
LIN {X 0,Y 608.422,Z 269.692,A -85,B 0,C 180,E1 -483.728,E2 -483.728} C_VEL
LIN {X 0,Y 608.438,Z 269.695,A -85,B 0,C 180,E1 -486.092,E2 -486.092} C_VEL
LIN {X 0,Y 608.463,Z 269.693,A -85,B 0,C 180,E1 -488.588,E2 -488.588} C_VEL
LIN {X 0,Y 608.439,Z 269.688,A -85,B 0,C 180,E1 -491.34,E2 -491.34} C_VEL
LIN {X 0,Y 608.444,Z 269.69,A -85,B 0,C 180,E1 -493.871,E2 -493.871} C_VEL
LIN {X 0,Y 608.477,Z 269.691,A -85,B 0,C 180,E1 -496.69,E2 -496.69} C_VEL
LIN {X 0,Y 608.463,Z 269.691,A -85,B 0,C 180,E1 -498.824,E2 -498.824} C_VEL
LIN {X 0,Y 608.434,Z 269.689,A -85,B 0,C 180,E1 -501.409,E2 -501.409} C_VEL
LIN {X 0,Y 608.437,Z 269.691,A -85,B 0,C 180,E1 -503.955,E2 -503.955} C_VEL
LIN {X 0,Y 608.444,Z 269.694,A -85,B 0,C 180,E1 -506.328,E2 -506.328} C_VEL
LIN {X 0,Y 608.475,Z 269.693,A -85,B 0,C 180,E1 -508.727,E2 -508.727} C_VEL
LIN {X 0,Y 608.47,Z 269.685,A -85,B 0,C 180,E1 -511.38,E2 -511.38} C_VEL
LIN {X 0,Y 608.434,Z 269.69,A -85,B 0,C 180,E1 -513.964,E2 -513.964} C_VEL
LIN {X 0,Y 608.451,Z 269.689,A -85,B 0,C 180,E1 -516.154,E2 -516.154} C_VEL
LIN {X 0,Y 608.463,Z 269.69,A -85,B 0,C 180,E1 -518.308,E2 -518.308} C_VEL
LIN {X 0,Y 608.47,Z 269.687,A -85,B 0,C 180,E1 -521.283,E2 -521.283} C_VEL
LIN {X 0,Y 608.454,Z 269.687,A -85,B 0,C 180,E1 -523.906,E2 -523.906} C_VEL
LIN {X 0,Y 608.468,Z 269.693,A -85,B 0,C 180,E1 -526.644,E2 -526.644} C_VEL
LIN {X 0,Y 608.46,Z 269.688,A -85,B 0,C 180,E1 -529.35,E2 -529.35} C_VEL
LIN {X 0,Y 608.472,Z 269.685,A -85,B 0,C 180,E1 -532.033,E2 -532.033} C_VEL
LIN {X 0,Y 608.466,Z 269.693,A -85,B 0,C 180,E1 -534.698,E2 -534.698} C_VEL
LIN {X 0,Y 608.467,Z 269.689,A -85,B 0,C 180,E1 -537.352,E2 -537.352} C_VEL
LIN {X 0,Y 608.476,Z 269.684,A -85,B 0,C 180,E1 -540,E2 -540} C_VEL
LIN {X 0,Y 608.473,Z 269.69,A -85,B 0,C 180,E1 -542.648,E2 -542.648} C_VEL
LIN {X 0,Y 608.458,Z 269.691,A -85,B 0,C 180,E1 -545.302,E2 -545.302} C_VEL
LIN {X 0,Y 608.469,Z 269.685,A -85,B 0,C 180,E1 -547.967,E2 -547.967} C_VEL
LIN {X 0,Y 608.452,Z 269.691,A -85,B 0,C 180,E1 -549.458,E2 -549.458} C_VEL
LIN {X 0,Y 607.768,Z 269.774,A -85,B 0,C 180,E1 -550.011,E2 -550.011} C_VEL
LIN {X 0,Y 604.911,Z 270.137,A -85,B 0,C 180,E1 -550.908,E2 -550.908} C_VEL
LIN {X 0,Y 602.51,Z 270.431,A -85,B 0,C 180,E1 -551.629,E2 -551.629} C_VEL
LIN {X 0,Y 601.484,Z 270.555,A -85,B 0,C 180,E1 -552.186,E2 -552.186} C_VEL
LIN {X 0,Y 601.402,Z 270.566,A -85,B 0,C 180,E1 -552.375,E2 -552.375} C_VEL
LIN {X 0,Y 601.429,Z 270.569,A -85,B 0,C 180,E1 -554.897,E2 -554.897} C_VEL
LIN {X 0,Y 601.429,Z 270.571,A -85,B 0,C 180,E1 -556.986,E2 -556.986} C_VEL
LIN {X 0,Y 601.396,Z 270.567,A -85,B 0,C 180,E1 -559.81,E2 -559.81} C_VEL
LIN {X 0,Y 601.414,Z 270.566,A -85,B 0,C 180,E1 -562.606,E2 -562.606} C_VEL
LIN {X 0,Y 601.397,Z 270.571,A -85,B 0,C 180,E1 -564.879,E2 -564.879} C_VEL
LIN {X 0,Y 601.411,Z 270.572,A -85,B 0,C 180,E1 -567.363,E2 -567.363} C_VEL
LIN {X 0,Y 601.404,Z 270.573,A -85,B 0,C 180,E1 -569.394,E2 -569.394} C_VEL
LIN {X 0,Y 601.39,Z 270.57,A -85,B 0,C 180,E1 -571.728,E2 -571.728} C_VEL
LIN {X 0,Y 601.415,Z 270.564,A -85,B 0,C 180,E1 -574.12,E2 -574.12} C_VEL
LIN {X 0,Y 601.4,Z 270.566,A -85,B 0,C 180,E1 -576.584,E2 -576.584} C_VEL
LIN {X 0,Y 601.404,Z 270.572,A -85,B 0,C 180,E1 -579.532,E2 -579.532} C_VEL
LIN {X 0,Y 601.406,Z 270.569,A -85,B 0,C 180,E1 -581.767,E2 -581.767} C_VEL
LIN {X 0,Y 601.397,Z 270.566,A -85,B 0,C 180,E1 -584.533,E2 -584.533} C_VEL
LIN {X 0,Y 601.405,Z 270.576,A -85,B 0,C 180,E1 -587.411,E2 -587.411} C_VEL
LIN {X 0,Y 601.395,Z 270.568,A -85,B 0,C 180,E1 -590.004,E2 -590.004} C_VEL
LIN {X 0,Y 601.395,Z 270.566,A -85,B 0,C 180,E1 -592.624,E2 -592.624} C_VEL
LIN {X 0,Y 601.409,Z 270.568,A -85,B 0,C 180,E1 -595.068,E2 -595.068} C_VEL
LIN {X 0,Y 601.432,Z 270.572,A -85,B 0,C 180,E1 -597.485,E2 -597.485} C_VEL
LIN {X 0,Y 601.4,Z 270.571,A -85,B 0,C 180,E1 -599.857,E2 -599.857} C_VEL
LIN {X 0,Y 601.365,Z 270.573,A -85,B 0,C 180,E1 -602.13,E2 -602.13} C_VEL
LIN {X 0,Y 601.419,Z 270.774,A -85,B 0,C 180,E1 -602.935,E2 -602.935} C_VEL
LIN {X 0,Y 601.435,Z 287.143,A -85,B 0,C 180,E1 -605.859,E2 -605.859} C_VEL
LIN {X 0,Y 601.408,Z 298.627,A -85,B 0,C 180,E1 -607.885,E2 -607.885} C_VEL
LIN {X 0,Y 601.668,Z 304.082,A -85,B 0,C 180,E1 -607.962,E2 -607.962} C_VEL
LIN {X 0,Y 601.594,Z 405.699,A -85,B 0,C 180,E1 -609.198,E2 -609.198} C_VEL
LIN {X 0,Y 601.574,Z 419.042,A -85,B 0,C 180,E1 -609.506,E2 -609.506} C_VEL
LIN {X 0,Y 601.562,Z 431.448,A -85,B 0,C 180,E1 -609.929,E2 -609.929} C_VEL
LIN {X 0,Y 601.494,Z 443.007,A -85,B 0,C 180,E1 -610.461,E2 -610.461} C_VEL
LIN {X 0,Y 601.439,Z 455.051,A -85,B 0,C 180,E1 -611.177,E2 -611.177} C_VEL
LIN {X 0,Y 601.469,Z 465.569,A -85,B 0,C 180,E1 -611.963,E2 -611.963} C_VEL
LIN {X 0,Y 601.396,Z 475.017,A -85,B 0,C 180,E1 -612.838,E2 -612.838} C_VEL
LIN {X 0,Y 601.407,Z 484.162,A -85,B 0,C 180,E1 -613.887,E2 -613.887} C_VEL
LIN {X 0,Y 601.371,Z 491.394,A -85,B 0,C 180,E1 -614.929,E2 -614.929} C_VEL
LIN {X 0,Y 601.353,Z 496.983,A -85,B 0,C 180,E1 -615.937,E2 -615.937} C_VEL
LIN {X 0,Y 601.333,Z 502.216,A -85,B 0,C 180,E1 -617.17,E2 -617.17} C_VEL
LIN {X 0,Y 601.367,Z 504.46,A -85,B 0,C 180,E1 -617.857,E2 -617.857} C_VEL
LIN {X 0,Y 601.337,Z 507.2,A -85,B 0,C 180,E1 -619.035,E2 -619.035} C_VEL
LIN {X 0,Y 601.328,Z 508.415,A -85,B 0,C 180,E1 -619.904,E2 -619.904} C_VEL
LIN {X 0,Y 601.335,Z 508.899,A -85,B 0,C 180,E1 -620.583,E2 -620.583} C_VEL
LIN {X 0,Y 601.332,Z 508.628,A -85,B 0,C 180,E1 -621.938,E2 -621.938} C_VEL
LIN {X 0,Y 601.321,Z 507.913,A -85,B 0,C 180,E1 -622.614,E2 -622.614} C_VEL
LIN {X 0,Y 601.349,Z 506.479,A -85,B 0,C 180,E1 -623.418,E2 -623.418} C_VEL
LIN {X 0,Y 601.352,Z 503.197,A -85,B 0,C 180,E1 -624.636,E2 -624.636} C_VEL
LIN {X 0,Y 601.355,Z 499.347,A -85,B 0,C 180,E1 -625.644,E2 -625.644} C_VEL
LIN {X 0,Y 601.353,Z 494.383,A -85,B 0,C 180,E1 -626.65,E2 -626.65} C_VEL
LIN {X 0,Y 601.394,Z 488.162,A -85,B 0,C 180,E1 -627.656,E2 -627.656} C_VEL
LIN {X 0,Y 601.406,Z 480.42,A -85,B 0,C 180,E1 -628.661,E2 -628.661} C_VEL
LIN {X 0,Y 601.415,Z 470.791,A -85,B 0,C 180,E1 -629.666,E2 -629.666} C_VEL
LIN {X 0,Y 601.45,Z 460.838,A -85,B 0,C 180,E1 -630.503,E2 -630.503} C_VEL
LIN {X 0,Y 601.441,Z 449.655,A -85,B 0,C 180,E1 -631.256,E2 -631.256} C_VEL
LIN {X 0,Y 601.498,Z 438.721,A -85,B 0,C 180,E1 -631.842,E2 -631.842} C_VEL
LIN {X 0,Y 601.535,Z 426.621,A -85,B 0,C 180,E1 -632.344,E2 -632.344} C_VEL
LIN {X 0,Y 601.552,Z 413.904,A -85,B 0,C 180,E1 -632.721,E2 -632.721} C_VEL
LIN {X 0,Y 601.569,Z 400.486,A -85,B 0,C 180,E1 -632.972,E2 -632.972} C_VEL
LIN {X 0,Y 601.626,Z 300.081,A -85,B 0,C 180,E1 -634.177,E2 -634.177} C_VEL
LIN {X 0,Y 601.408,Z 298.478,A -85,B 0,C 180,E1 -634.231,E2 -634.231} C_VEL
LIN {X 0,Y 601.463,Z 282.54,A -85,B 0,C 180,E1 -637.048,E2 -637.048} C_VEL
LIN {X 0,Y 601.402,Z 270.568,A -85,B 0,C 180,E1 -639.205,E2 -639.205} C_VEL
LIN {X 0,Y 601.402,Z 270.569,A -85,B 0,C 180,E1 -642.143,E2 -642.143} C_VEL
LIN {X 0,Y 601.417,Z 270.57,A -85,B 0,C 180,E1 -644.898,E2 -644.898} C_VEL
LIN {X 0,Y 601.406,Z 270.57,A -85,B 0,C 180,E1 -646.987,E2 -646.987} C_VEL
LIN {X 0,Y 601.378,Z 270.568,A -85,B 0,C 180,E1 -649.811,E2 -649.811} C_VEL
LIN {X 0,Y 601.381,Z 270.568,A -85,B 0,C 180,E1 -651.961,E2 -651.961} C_VEL
LIN {X 0,Y 601.384,Z 270.579,A -85,B 0,C 180,E1 -654.88,E2 -654.88} C_VEL
LIN {X 0,Y 601.387,Z 270.57,A -85,B 0,C 180,E1 -657.356,E2 -657.356} C_VEL
LIN {X 0,Y 601.378,Z 270.572,A -85,B 0,C 180,E1 -659.396,E2 -659.396} C_VEL
LIN {X 0,Y 601.385,Z 270.568,A -85,B 0,C 180,E1 -661.728,E2 -661.728} C_VEL
LIN {X 0,Y 601.41,Z 270.564,A -85,B 0,C 180,E1 -664.12,E2 -664.12} C_VEL
LIN {X 0,Y 601.437,Z 270.567,A -85,B 0,C 180,E1 -667.381,E2 -667.381} C_VEL
LIN {X 0,Y 601.38,Z 270.568,A -85,B 0,C 180,E1 -669.998,E2 -669.998} C_VEL
LIN {X 0,Y 601.379,Z 270.57,A -85,B 0,C 180,E1 -672.674,E2 -672.674} C_VEL
LIN {X 0,Y 601.405,Z 270.573,A -85,B 0,C 180,E1 -675.479,E2 -675.479} C_VEL
LIN {X 0,Y 601.402,Z 270.565,A -85,B 0,C 180,E1 -678.41,E2 -678.41} C_VEL
LIN {X 0,Y 601.392,Z 270.568,A -85,B 0,C 180,E1 -680.871,E2 -680.871} C_VEL
LIN {X 0,Y 601.391,Z 270.573,A -85,B 0,C 180,E1 -683.741,E2 -683.741} C_VEL
LIN {X 0,Y 601.408,Z 270.567,A -85,B 0,C 180,E1 -686.069,E2 -686.069} C_VEL
LIN {X 0,Y 601.41,Z 270.564,A -85,B 0,C 180,E1 -688.548,E2 -688.548} C_VEL
LIN {X 0,Y 601.433,Z 270.567,A -85,B 0,C 180,E1 -691.373,E2 -691.373} C_VEL
LIN {X 0,Y 601.379,Z 270.569,A -85,B 0,C 180,E1 -694.38,E2 -694.38} C_VEL
LIN {X 0,Y 601.369,Z 270.569,A -85,B 0,C 180,E1 -696.587,E2 -696.587} C_VEL
LIN {X 0,Y 601.428,Z 270.566,A -85,B 0,C 180,E1 -699.478,E2 -699.478} C_VEL
LIN {X 0,Y 601.37,Z 270.573,A -85,B 0,C 180,E1 -702.311,E2 -702.311} C_VEL
LIN {X 0,Y 601.385,Z 270.57,A -85,B 0,C 180,E1 -704.408,E2 -704.408} C_VEL
LIN {X 0,Y 601.39,Z 270.569,A -85,B 0,C 180,E1 -706.483,E2 -706.483} C_VEL
LIN {X 0,Y 601.358,Z 270.57,A -85,B 0,C 180,E1 -709.023,E2 -709.023} C_VEL
LIN {X 0,Y 601.387,Z 270.567,A -85,B 0,C 180,E1 -711.261,E2 -711.261} C_VEL
LIN {X 0,Y 601.415,Z 270.571,A -85,B 0,C 180,E1 -713.963,E2 -713.963} C_VEL
LIN {X 0,Y 601.369,Z 270.573,A -85,B 0,C 180,E1 -716.65,E2 -716.65} C_VEL
LIN {X 0,Y 601.392,Z 270.57,A -85,B 0,C 180,E1 -718.661,E2 -718.661} C_VEL
LIN {X 0,Y 601.426,Z 270.567,A -85,B 0,C 180,E1 -720.669,E2 -720.669} C_VEL
LIN {X 0,Y 601.357,Z 270.57,A -85,B 0,C 180,E1 -723.35,E2 -723.35} C_VEL
LIN {X 0,Y 601.397,Z 270.57,A -85,B 0,C 180,E1 -726.037,E2 -726.037} C_VEL
LIN {X 0,Y 601.402,Z 270.571,A -85,B 0,C 180,E1 -728.738,E2 -728.738} C_VEL
LIN {X 0,Y 601.374,Z 270.568,A -85,B 0,C 180,E1 -731.459,E2 -731.459} C_VEL
LIN {X 0,Y 601.405,Z 270.569,A -85,B 0,C 180,E1 -734.206,E2 -734.206} C_VEL
LIN {X 0,Y 601.405,Z 270.57,A -85,B 0,C 180,E1 -736.987,E2 -736.987} C_VEL
LIN {X 0,Y 601.376,Z 270.568,A -85,B 0,C 180,E1 -739.81,E2 -739.81} C_VEL
LIN {X 0,Y 601.385,Z 270.567,A -85,B 0,C 180,E1 -741.96,E2 -741.96} C_VEL
LIN {X 0,Y 601.382,Z 270.578,A -85,B 0,C 180,E1 -744.879,E2 -744.879} C_VEL
LIN {X 0,Y 601.383,Z 270.57,A -85,B 0,C 180,E1 -747.356,E2 -747.356} C_VEL
LIN {X 0,Y 601.375,Z 270.572,A -85,B 0,C 180,E1 -749.395,E2 -749.395} C_VEL
LIN {X 0,Y 601.382,Z 270.568,A -85,B 0,C 180,E1 -751.728,E2 -751.728} C_VEL
LIN {X 0,Y 601.408,Z 270.564,A -85,B 0,C 180,E1 -754.12,E2 -754.12} C_VEL
LIN {X 0,Y 601.434,Z 270.567,A -85,B 0,C 180,E1 -757.381,E2 -757.381} C_VEL
LIN {X 0,Y 601.377,Z 270.568,A -85,B 0,C 180,E1 -759.998,E2 -759.998} C_VEL
LIN {X 0,Y 601.378,Z 270.57,A -85,B 0,C 180,E1 -762.673,E2 -762.673} C_VEL
LIN {X 0,Y 601.402,Z 270.572,A -85,B 0,C 180,E1 -765.479,E2 -765.479} C_VEL
LIN {X 0,Y 601.399,Z 270.565,A -85,B 0,C 180,E1 -768.41,E2 -768.41} C_VEL
LIN {X 0,Y 601.391,Z 270.569,A -85,B 0,C 180,E1 -770.871,E2 -770.871} C_VEL
LIN {X 0,Y 601.389,Z 270.573,A -85,B 0,C 180,E1 -773.741,E2 -773.741} C_VEL
LIN {X 0,Y 601.406,Z 270.567,A -85,B 0,C 180,E1 -776.068,E2 -776.068} C_VEL
LIN {X 0,Y 601.407,Z 270.564,A -85,B 0,C 180,E1 -778.548,E2 -778.548} C_VEL
LIN {X 0,Y 601.432,Z 270.568,A -85,B 0,C 180,E1 -781.373,E2 -781.373} C_VEL
LIN {X 0,Y 601.376,Z 270.57,A -85,B 0,C 180,E1 -784.379,E2 -784.379} C_VEL
LIN {X 0,Y 601.39,Z 270.648,A -85,B 0,C 180,E1 -786.748,E2 -786.748} C_VEL
LIN {X 0,Y 601.713,Z 275.67,A -85,B 0,C 180,E1 -787.447,E2 -787.447} C_VEL
LIN {X 0,Y 601.583,Z 296.076,A -85,B 0,C 180,E1 -790.196,E2 -790.196} C_VEL
LIN {X 0,Y 601.524,Z 314.691,A -85,B 0,C 180,E1 -792.666,E2 -792.666} C_VEL
LIN {X 0,Y 601.506,Z 337.294,A -85,B 0,C 180,E1 -795.624,E2 -795.624} C_VEL
LIN {X 0,Y 601.429,Z 346.518,A -85,B 0,C 180,E1 -796.817,E2 -796.817} C_VEL
LIN {X 0,Y 601.643,Z 356.05,A -85,B 0,C 180,E1 -796.94,E2 -796.94} C_VEL
LIN {X 0,Y 601.591,Z 454.924,A -85,B 0,C 180,E1 -798.139,E2 -798.139} C_VEL
LIN {X 0,Y 601.554,Z 468.202,A -85,B 0,C 180,E1 -798.437,E2 -798.437} C_VEL
LIN {X 0,Y 601.54,Z 480.645,A -85,B 0,C 180,E1 -798.853,E2 -798.853} C_VEL
LIN {X 0,Y 601.519,Z 492.625,A -85,B 0,C 180,E1 -799.396,E2 -799.396} C_VEL
LIN {X 0,Y 601.477,Z 504.192,A -85,B 0,C 180,E1 -800.075,E2 -800.075} C_VEL
LIN {X 0,Y 601.444,Z 514.59,A -85,B 0,C 180,E1 -800.838,E2 -800.838} C_VEL
LIN {X 0,Y 601.429,Z 523.107,A -85,B 0,C 180,E1 -801.6,E2 -801.6} C_VEL
LIN {X 0,Y 601.418,Z 530.957,A -85,B 0,C 180,E1 -802.445,E2 -802.445} C_VEL
LIN {X 0,Y 601.37,Z 538.221,A -85,B 0,C 180,E1 -803.397,E2 -803.397} C_VEL
LIN {X 0,Y 601.372,Z 543.864,A -85,B 0,C 180,E1 -804.299,E2 -804.299} C_VEL
LIN {X 0,Y 601.336,Z 548.948,A -85,B 0,C 180,E1 -805.307,E2 -805.307} C_VEL
LIN {X 0,Y 601.368,Z 552.895,A -85,B 0,C 180,E1 -806.314,E2 -806.314} C_VEL
LIN {X 0,Y 601.325,Z 555.808,A -85,B 0,C 180,E1 -807.32,E2 -807.32} C_VEL
LIN {X 0,Y 601.342,Z 557.201,A -85,B 0,C 180,E1 -807.99,E2 -807.99} C_VEL
LIN {X 0,Y 601.339,Z 558.783,A -85,B 0,C 180,E1 -809.33,E2 -809.33} C_VEL
LIN {X 0,Y 601.335,Z 559,A -85,B 0,C 180,E1 -810,E2 -810} C_VEL
LIN {X 0,Y 601.347,Z 558.185,A -85,B 0,C 180,E1 -811.339,E2 -811.339} C_VEL
LIN {X 0,Y 601.342,Z 557.203,A -85,B 0,C 180,E1 -812.009,E2 -812.009} C_VEL
LIN {X 0,Y 601.325,Z 555.81,A -85,B 0,C 180,E1 -812.679,E2 -812.679} C_VEL
LIN {X 0,Y 601.367,Z 552.897,A -85,B 0,C 180,E1 -813.685,E2 -813.685} C_VEL
LIN {X 0,Y 601.336,Z 548.952,A -85,B 0,C 180,E1 -814.692,E2 -814.692} C_VEL
LIN {X 0,Y 601.372,Z 542.88,A -85,B 0,C 180,E1 -815.869,E2 -815.869} C_VEL
LIN {X 0,Y 601.381,Z 536.239,A -85,B 0,C 180,E1 -816.879,E2 -816.879} C_VEL
LIN {X 0,Y 601.4,Z 527.993,A -85,B 0,C 180,E1 -817.892,E2 -817.892} C_VEL
LIN {X 0,Y 601.436,Z 519.542,A -85,B 0,C 180,E1 -818.737,E2 -818.737} C_VEL
LIN {X 0,Y 601.444,Z 509.098,A -85,B 0,C 180,E1 -819.585,E2 -819.585} C_VEL
LIN {X 0,Y 601.481,Z 498.765,A -85,B 0,C 180,E1 -820.264,E2 -820.264} C_VEL
LIN {X 0,Y 601.538,Z 486.596,A -85,B 0,C 180,E1 -820.896,E2 -820.896} C_VEL
LIN {X 0,Y 601.543,Z 474.229,A -85,B 0,C 180,E1 -821.379,E2 -821.379} C_VEL
LIN {X 0,Y 601.557,Z 461.456,A -85,B 0,C 180,E1 -821.733,E2 -821.733} C_VEL
LIN {X 0,Y 601.596,Z 449.117,A -85,B 0,C 180,E1 -821.946,E2 -821.946} C_VEL
LIN {X 0,Y 601.508,Z 347.179,A -85,B 0,C 180,E1 -823.169,E2 -823.169} C_VEL
LIN {X 0,Y 601.447,Z 346.276,A -85,B 0,C 180,E1 -823.214,E2 -823.214} C_VEL
LIN {X 0,Y 601.467,Z 326.664,A -85,B 0,C 180,E1 -825.763,E2 -825.763} C_VEL
LIN {X 0,Y 601.59,Z 304.942,A -85,B 0,C 180,E1 -828.622,E2 -828.622} C_VEL
LIN {X 0,Y 601.628,Z 284.117,A -85,B 0,C 180,E1 -831.41,E2 -831.41} C_VEL
LIN {X 0,Y 601.652,Z 272.15,A -85,B 0,C 180,E1 -833.036,E2 -833.036} C_VEL
LIN {X 0,Y 601.379,Z 270.572,A -85,B 0,C 180,E1 -833.275,E2 -833.275} C_VEL
LIN {X 0,Y 601.378,Z 270.57,A -85,B 0,C 180,E1 -835.619,E2 -835.619} C_VEL
LIN {X 0,Y 601.432,Z 270.567,A -85,B 0,C 180,E1 -838.626,E2 -838.626} C_VEL
LIN {X 0,Y 601.408,Z 270.565,A -85,B 0,C 180,E1 -841.452,E2 -841.452} C_VEL
LIN {X 0,Y 601.411,Z 270.571,A -85,B 0,C 180,E1 -844.119,E2 -844.119} C_VEL
LIN {X 0,Y 601.427,Z 270.562,A -85,B 0,C 180,E1 -847.381,E2 -847.381} C_VEL
LIN {X 0,Y 601.394,Z 270.57,A -85,B 0,C 180,E1 -849.996,E2 -849.996} C_VEL
LIN {X 0,Y 601.411,Z 270.571,A -85,B 0,C 180,E1 -852.67,E2 -852.67} C_VEL
LIN {X 0,Y 601.396,Z 270.566,A -85,B 0,C 180,E1 -855.479,E2 -855.479} C_VEL
LIN {X 0,Y 601.421,Z 270.572,A -85,B 0,C 180,E1 -858.407,E2 -858.407} C_VEL
LIN {X 0,Y 601.428,Z 270.567,A -85,B 0,C 180,E1 -860.875,E2 -860.875} C_VEL
LIN {X 0,Y 601.4,Z 270.566,A -85,B 0,C 180,E1 -863.417,E2 -863.417} C_VEL
LIN {X 0,Y 601.413,Z 270.566,A -85,B 0,C 180,E1 -866.066,E2 -866.066} C_VEL
LIN {X 0,Y 601.437,Z 270.571,A -85,B 0,C 180,E1 -868.542,E2 -868.542} C_VEL
LIN {X 0,Y 601.43,Z 270.562,A -85,B 0,C 180,E1 -871.373,E2 -871.373} C_VEL
LIN {X 0,Y 601.396,Z 270.566,A -85,B 0,C 180,E1 -873.636,E2 -873.636} C_VEL
LIN {X 0,Y 601.412,Z 270.573,A -85,B 0,C 180,E1 -876.589,E2 -876.589} C_VEL
LIN {X 0,Y 601.431,Z 270.562,A -85,B 0,C 180,E1 -879.478,E2 -879.478} C_VEL
LIN {X 0,Y 601.394,Z 270.57,A -85,B 0,C 180,E1 -882.312,E2 -882.312} C_VEL
LIN {X 0,Y 601.411,Z 270.568,A -85,B 0,C 180,E1 -884.409,E2 -884.409} C_VEL
LIN {X 0,Y 601.421,Z 270.567,A -85,B 0,C 180,E1 -887.172,E2 -887.172} C_VEL
LIN {X 0,Y 601.426,Z 270.562,A -85,B 0,C 180,E1 -889.905,E2 -889.905} C_VEL
LIN {X 0,Y 601.439,Z 270.567,A -85,B 0,C 180,E1 -892.615,E2 -892.615} C_VEL
LIN {X 0,Y 601.413,Z 270.567,A -85,B 0,C 180,E1 -895.308,E2 -895.308} C_VEL
LIN {X 0,Y 601.431,Z 270.561,A -85,B 0,C 180,E1 -897.991,E2 -897.991} C_VEL
LIN {X 0,Y 601.448,Z 270.565,A -85,B 0,C 180,E1 -900.67,E2 -900.67} C_VEL
LIN {X 0,Y 601.422,Z 270.567,A -85,B 0,C 180,E1 -903.35,E2 -903.35} C_VEL
LIN {X 0,Y 601.407,Z 270.564,A -85,B 0,C 180,E1 -906.037,E2 -906.037} C_VEL
LIN {X 0,Y 601.433,Z 270.567,A -85,B 0,C 180,E1 -908.738,E2 -908.738} C_VEL
LIN {X 0,Y 601.429,Z 270.566,A -85,B 0,C 180,E1 -911.458,E2 -911.458} C_VEL
LIN {X 0,Y 601.402,Z 270.566,A -85,B 0,C 180,E1 -912.375,E2 -912.375} C_VEL
LIN {X 0,Y 600.743,Z 270.656,A -85,B 0,C 180,E1 -912.934,E2 -912.934} C_VEL
LIN {X 0,Y 597.896,Z 271.015,A -85,B 0,C 180,E1 -913.842,E2 -913.842} C_VEL
LIN {X 0,Y 595.484,Z 271.316,A -85,B 0,C 180,E1 -914.572,E2 -914.572} C_VEL
LIN {X 0,Y 594.444,Z 271.442,A -85,B 0,C 180,E1 -915.136,E2 -915.136} C_VEL
LIN {X 0,Y 594.358,Z 271.449,A -85,B 0,C 180,E1 -915.326,E2 -915.326} C_VEL
LIN {X 0,Y 594.385,Z 271.449,A -85,B 0,C 180,E1 -917.194,E2 -917.194} C_VEL
LIN {X 0,Y 594.369,Z 271.441,A -85,B 0,C 180,E1 -920.054,E2 -920.054} C_VEL
LIN {X 0,Y 594.353,Z 271.451,A -85,B 0,C 180,E1 -922.968,E2 -922.968} C_VEL
LIN {X 0,Y 594.366,Z 271.453,A -85,B 0,C 180,E1 -925.194,E2 -925.194} C_VEL
LIN {X 0,Y 594.366,Z 271.447,A -85,B 0,C 180,E1 -927.524,E2 -927.524} C_VEL
LIN {X 0,Y 594.366,Z 271.442,A -85,B 0,C 180,E1 -930.326,E2 -930.326} C_VEL
LIN {X 0,Y 594.374,Z 271.446,A -85,B 0,C 180,E1 -932.951,E2 -932.951} C_VEL
LIN {X 0,Y 594.352,Z 271.452,A -85,B 0,C 180,E1 -935.409,E2 -935.409} C_VEL
LIN {X 0,Y 594.369,Z 271.442,A -85,B 0,C 180,E1 -937.942,E2 -937.942} C_VEL
LIN {X 0,Y 594.375,Z 271.443,A -85,B 0,C 180,E1 -940.822,E2 -940.822} C_VEL
LIN {X 0,Y 594.343,Z 271.448,A -85,B 0,C 180,E1 -943.838,E2 -943.838} C_VEL
LIN {X 0,Y 594.349,Z 271.445,A -85,B 0,C 180,E1 -946.699,E2 -946.699} C_VEL
LIN {X 0,Y 594.356,Z 271.454,A -85,B 0,C 180,E1 -949.433,E2 -949.433} C_VEL
LIN {X 0,Y 594.355,Z 271.443,A -85,B 0,C 180,E1 -952.397,E2 -952.397} C_VEL
LIN {X 0,Y 594.375,Z 271.45,A -85,B 0,C 180,E1 -955.42,E2 -955.42} C_VEL
LIN {X 0,Y 594.361,Z 271.448,A -85,B 0,C 180,E1 -957.853,E2 -957.853} C_VEL
LIN {X 0,Y 594.344,Z 271.446,A -85,B 0,C 180,E1 -960.222,E2 -960.222} C_VEL
LIN {X 0,Y 594.344,Z 271.521,A -85,B 0,C 180,E1 -962.848,E2 -962.848} C_VEL
LIN {X 0,Y 594.422,Z 283.367,A -85,B 0,C 180,E1 -964.997,E2 -964.997} C_VEL
LIN {X 0,Y 594.359,Z 298.601,A -85,B 0,C 180,E1 -967.722,E2 -967.722} C_VEL
LIN {X 0,Y 594.756,Z 303.919,A -85,B 0,C 180,E1 -967.805,E2 -967.805} C_VEL
LIN {X 0,Y 594.665,Z 404.72,A -85,B 0,C 180,E1 -969.04,E2 -969.04} C_VEL
LIN {X 0,Y 594.609,Z 418.216,A -85,B 0,C 180,E1 -969.346,E2 -969.346} C_VEL
LIN {X 0,Y 594.579,Z 430.837,A -85,B 0,C 180,E1 -969.774,E2 -969.774} C_VEL
LIN {X 0,Y 594.505,Z 442.576,A -85,B 0,C 180,E1 -970.311,E2 -970.311} C_VEL
LIN {X 0,Y 594.438,Z 453.978,A -85,B 0,C 180,E1 -970.987,E2 -970.987} C_VEL
LIN {X 0,Y 594.424,Z 465.285,A -85,B 0,C 180,E1 -971.83,E2 -971.83} C_VEL
LIN {X 0,Y 594.37,Z 473.956,A -85,B 0,C 180,E1 -972.629,E2 -972.629} C_VEL
LIN {X 0,Y 594.315,Z 483.275,A -85,B 0,C 180,E1 -973.689,E2 -973.689} C_VEL
LIN {X 0,Y 594.307,Z 490.725,A -85,B 0,C 180,E1 -974.745,E2 -974.745} C_VEL
LIN {X 0,Y 594.265,Z 496.986,A -85,B 0,C 180,E1 -975.876,E2 -975.876} C_VEL
LIN {X 0,Y 594.259,Z 501.819,A -85,B 0,C 180,E1 -977.015,E2 -977.015} C_VEL
LIN {X 0,Y 594.258,Z 504.127,A -85,B 0,C 180,E1 -977.709,E2 -977.709} C_VEL
LIN {X 0,Y 594.252,Z 507.178,A -85,B 0,C 180,E1 -978.998,E2 -978.998} C_VEL
LIN {X 0,Y 594.23,Z 508.291,A -85,B 0,C 180,E1 -979.782,E2 -979.782} C_VEL
LIN {X 0,Y 594.255,Z 508.854,A -85,B 0,C 180,E1 -980.47,E2 -980.47} C_VEL
LIN {X 0,Y 594.227,Z 508.981,A -85,B 0,C 180,E1 -981.156,E2 -981.156} C_VEL
LIN {X 0,Y 594.247,Z 508.04,A -85,B 0,C 180,E1 -982.525,E2 -982.525} C_VEL
LIN {X 0,Y 594.264,Z 506.52,A -85,B 0,C 180,E1 -983.427,E2 -983.427} C_VEL
LIN {X 0,Y 594.265,Z 503.531,A -85,B 0,C 180,E1 -984.572,E2 -984.572} C_VEL
LIN {X 0,Y 594.271,Z 499.794,A -85,B 0,C 180,E1 -985.592,E2 -985.592} C_VEL
LIN {X 0,Y 594.275,Z 494.952,A -85,B 0,C 180,E1 -986.611,E2 -986.611} C_VEL
LIN {X 0,Y 594.302,Z 488.866,A -85,B 0,C 180,E1 -987.628,E2 -987.628} C_VEL
LIN {X 0,Y 594.34,Z 481.326,A -85,B 0,C 180,E1 -988.645,E2 -988.645} C_VEL
LIN {X 0,Y 594.366,Z 473.648,A -85,B 0,C 180,E1 -989.492,E2 -989.492} C_VEL
LIN {X 0,Y 594.42,Z 463.257,A -85,B 0,C 180,E1 -990.424,E2 -990.424} C_VEL
LIN {X 0,Y 594.419,Z 452.741,A -85,B 0,C 180,E1 -991.186,E2 -991.186} C_VEL
LIN {X 0,Y 594.483,Z 442.579,A -85,B 0,C 180,E1 -991.779,E2 -991.779} C_VEL
LIN {X 0,Y 594.553,Z 430.52,A -85,B 0,C 180,E1 -992.329,E2 -992.329} C_VEL
LIN {X 0,Y 594.595,Z 417.194,A -85,B 0,C 180,E1 -992.774,E2 -992.774} C_VEL
LIN {X 0,Y 594.608,Z 404.836,A -85,B 0,C 180,E1 -993.049,E2 -993.049} C_VEL
LIN {X 0,Y 594.624,Z 300.252,A -85,B 0,C 180,E1 -994.332,E2 -994.332} C_VEL
LIN {X 0,Y 594.358,Z 298.614,A -85,B 0,C 180,E1 -994.366,E2 -994.366} C_VEL
LIN {X 0,Y 594.438,Z 283.154,A -85,B 0,C 180,E1 -997.132,E2 -997.132} C_VEL
LIN {X 0,Y 594.357,Z 271.446,A -85,B 0,C 180,E1 -999.272,E2 -999.272} C_VEL
LIN {X 0,Y 594.379,Z 271.446,A -85,B 0,C 180,E1 -1002.289,E2 -1002.289} C_VEL
LIN {X 0,Y 594.358,Z 271.446,A -85,B 0,C 180,E1 -1005.079,E2 -1005.079} C_VEL
LIN {X 0,Y 594.342,Z 271.447,A -85,B 0,C 180,E1 -1007.195,E2 -1007.195} C_VEL
LIN {X 0,Y 594.356,Z 271.445,A -85,B 0,C 180,E1 -1009.335,E2 -1009.335} C_VEL
LIN {X 0,Y 594.348,Z 271.444,A -85,B 0,C 180,E1 -1011.504,E2 -1011.504} C_VEL
LIN {X 0,Y 594.353,Z 271.443,A -85,B 0,C 180,E1 -1013.706,E2 -1013.706} C_VEL
LIN {X 0,Y 594.367,Z 271.449,A -85,B 0,C 180,E1 -1016.701,E2 -1016.701} C_VEL
LIN {X 0,Y 594.377,Z 271.451,A -85,B 0,C 180,E1 -1018.999,E2 -1018.999} C_VEL
LIN {X 0,Y 594.36,Z 271.444,A -85,B 0,C 180,E1 -1021.639,E2 -1021.639} C_VEL
LIN {X 0,Y 594.364,Z 271.442,A -85,B 0,C 180,E1 -1024.135,E2 -1024.135} C_VEL
LIN {X 0,Y 594.384,Z 271.45,A -85,B 0,C 180,E1 -1027.087,E2 -1027.087} C_VEL
LIN {X 0,Y 594.34,Z 271.447,A -85,B 0,C 180,E1 -1029.769,E2 -1029.769} C_VEL
LIN {X 0,Y 594.338,Z 271.445,A -85,B 0,C 180,E1 -1032.379,E2 -1032.379} C_VEL
LIN {X 0,Y 594.343,Z 271.453,A -85,B 0,C 180,E1 -1035.194,E2 -1035.194} C_VEL
LIN {X 0,Y 594.361,Z 271.443,A -85,B 0,C 180,E1 -1038.155,E2 -1038.155} C_VEL
LIN {X 0,Y 594.351,Z 271.443,A -85,B 0,C 180,E1 -1040.317,E2 -1040.317} C_VEL
LIN {X 0,Y 594.355,Z 271.445,A -85,B 0,C 180,E1 -1042.911,E2 -1042.911} C_VEL
LIN {X 0,Y 594.368,Z 271.447,A -85,B 0,C 180,E1 -1045.864,E2 -1045.864} C_VEL
LIN {X 0,Y 594.358,Z 271.442,A -85,B 0,C 180,E1 -1048.649,E2 -1048.649} C_VEL
LIN {X 0,Y 594.381,Z 271.441,A -85,B 0,C 180,E1 -1051.044,E2 -1051.044} C_VEL
LIN {X 0,Y 594.343,Z 271.449,A -85,B 0,C 180,E1 -1054.054,E2 -1054.054} C_VEL
LIN {X 0,Y 594.36,Z 271.445,A -85,B 0,C 180,E1 -1056.294,E2 -1056.294} C_VEL
LIN {X 0,Y 594.4,Z 271.439,A -85,B 0,C 180,E1 -1059.224,E2 -1059.224} C_VEL
LIN {X 0,Y 594.328,Z 271.454,A -85,B 0,C 180,E1 -1062.094,E2 -1062.094} C_VEL
LIN {X 0,Y 594.343,Z 271.45,A -85,B 0,C 180,E1 -1064.218,E2 -1064.218} C_VEL
LIN {X 0,Y 594.364,Z 271.447,A -85,B 0,C 180,E1 -1066.32,E2 -1066.32} C_VEL
LIN {X 0,Y 594.335,Z 271.445,A -85,B 0,C 180,E1 -1068.956,E2 -1068.956} C_VEL
LIN {X 0,Y 594.378,Z 271.446,A -85,B 0,C 180,E1 -1071.843,E2 -1071.843} C_VEL
LIN {X 0,Y 594.364,Z 271.446,A -85,B 0,C 180,E1 -1074.572,E2 -1074.572} C_VEL
LIN {X 0,Y 594.37,Z 271.441,A -85,B 0,C 180,E1 -1077.289,E2 -1077.289} C_VEL
LIN {X 0,Y 594.414,Z 271.441,A -85,B 0,C 180,E1 -1080,E2 -1080} C_VEL
LIN {X 0,Y 594.384,Z 271.444,A -85,B 0,C 180,E1 -1082.711,E2 -1082.711} C_VEL
LIN {X 0,Y 594.353,Z 271.443,A -85,B 0,C 180,E1 -1085.428,E2 -1085.428} C_VEL
LIN {X 0,Y 594.357,Z 271.448,A -85,B 0,C 180,E1 -1088.157,E2 -1088.157} C_VEL
LIN {X 0,Y 594.334,Z 271.448,A -85,B 0,C 180,E1 -1091.044,E2 -1091.044} C_VEL
LIN {X 0,Y 594.344,Z 271.444,A -85,B 0,C 180,E1 -1093.68,E2 -1093.68} C_VEL
LIN {X 0,Y 594.4,Z 271.445,A -85,B 0,C 180,E1 -1096.485,E2 -1096.485} C_VEL
LIN {X 0,Y 594.353,Z 271.445,A -85,B 0,C 180,E1 -1099.335,E2 -1099.335} C_VEL
LIN {X 0,Y 594.347,Z 271.444,A -85,B 0,C 180,E1 -1101.504,E2 -1101.504} C_VEL
LIN {X 0,Y 594.351,Z 271.443,A -85,B 0,C 180,E1 -1103.706,E2 -1103.706} C_VEL
LIN {X 0,Y 594.356,Z 271.451,A -85,B 0,C 180,E1 -1106.701,E2 -1106.701} C_VEL
LIN {X 0,Y 594.374,Z 271.45,A -85,B 0,C 180,E1 -1108.999,E2 -1108.999} C_VEL
LIN {X 0,Y 594.357,Z 271.444,A -85,B 0,C 180,E1 -1111.639,E2 -1111.639} C_VEL
LIN {X 0,Y 594.362,Z 271.442,A -85,B 0,C 180,E1 -1114.135,E2 -1114.135} C_VEL
LIN {X 0,Y 594.381,Z 271.451,A -85,B 0,C 180,E1 -1117.087,E2 -1117.087} C_VEL
LIN {X 0,Y 594.337,Z 271.447,A -85,B 0,C 180,E1 -1119.769,E2 -1119.769} C_VEL
LIN {X 0,Y 594.336,Z 271.445,A -85,B 0,C 180,E1 -1122.378,E2 -1122.378} C_VEL
LIN {X 0,Y 594.341,Z 271.454,A -85,B 0,C 180,E1 -1125.194,E2 -1125.194} C_VEL
LIN {X 0,Y 594.358,Z 271.443,A -85,B 0,C 180,E1 -1128.155,E2 -1128.155} C_VEL
LIN {X 0,Y 594.349,Z 271.444,A -85,B 0,C 180,E1 -1130.317,E2 -1130.317} C_VEL
LIN {X 0,Y 594.353,Z 271.445,A -85,B 0,C 180,E1 -1132.91,E2 -1132.91} C_VEL
LIN {X 0,Y 594.367,Z 271.446,A -85,B 0,C 180,E1 -1135.864,E2 -1135.864} C_VEL
LIN {X 0,Y 594.356,Z 271.443,A -85,B 0,C 180,E1 -1138.648,E2 -1138.648} C_VEL
LIN {X 0,Y 594.379,Z 271.442,A -85,B 0,C 180,E1 -1141.043,E2 -1141.043} C_VEL
LIN {X 0,Y 594.341,Z 271.45,A -85,B 0,C 180,E1 -1144.054,E2 -1144.054} C_VEL
LIN {X 0,Y 594.335,Z 271.479,A -85,B 0,C 180,E1 -1146.57,E2 -1146.57} C_VEL
LIN {X 0,Y 594.798,Z 275.642,A -85,B 0,C 180,E1 -1147.166,E2 -1147.166} C_VEL
LIN {X 0,Y 594.685,Z 294.747,A -85,B 0,C 180,E1 -1149.776,E2 -1149.776} C_VEL
LIN {X 0,Y 594.558,Z 316.02,A -85,B 0,C 180,E1 -1152.634,E2 -1152.634} C_VEL
LIN {X 0,Y 594.489,Z 338.624,A -85,B 0,C 180,E1 -1155.625,E2 -1155.625} C_VEL
LIN {X 0,Y 594.436,Z 346.435,A -85,B 0,C 180,E1 -1156.648,E2 -1156.648} C_VEL
LIN {X 0,Y 594.758,Z 352.472,A -85,B 0,C 180,E1 -1156.743,E2 -1156.743} C_VEL
LIN {X 0,Y 594.643,Z 454.923,A -85,B 0,C 180,E1 -1157.998,E2 -1157.998} C_VEL
LIN {X 0,Y 594.619,Z 468.203,A -85,B 0,C 180,E1 -1158.3,E2 -1158.3} C_VEL
LIN {X 0,Y 594.595,Z 480.434,A -85,B 0,C 180,E1 -1158.713,E2 -1158.713} C_VEL
LIN {X 0,Y 594.533,Z 492.624,A -85,B 0,C 180,E1 -1159.27,E2 -1159.27} C_VEL
LIN {X 0,Y 594.471,Z 504.194,A -85,B 0,C 180,E1 -1159.957,E2 -1159.957} C_VEL
LIN {X 0,Y 594.414,Z 514.591,A -85,B 0,C 180,E1 -1160.729,E2 -1160.729} C_VEL
LIN {X 0,Y 594.383,Z 523.108,A -85,B 0,C 180,E1 -1161.5,E2 -1161.5} C_VEL
LIN {X 0,Y 594.347,Z 530.957,A -85,B 0,C 180,E1 -1162.355,E2 -1162.355} C_VEL
LIN {X 0,Y 594.283,Z 538.809,A -85,B 0,C 180,E1 -1163.408,E2 -1163.408} C_VEL
LIN {X 0,Y 594.289,Z 545.678,A -85,B 0,C 180,E1 -1164.571,E2 -1164.571} C_VEL
LIN {X 0,Y 594.27,Z 550.37,A -85,B 0,C 180,E1 -1165.591,E2 -1165.591} C_VEL
LIN {X 0,Y 594.267,Z 553.955,A -85,B 0,C 180,E1 -1166.61,E2 -1166.61} C_VEL
LIN {X 0,Y 594.226,Z 555.808,A -85,B 0,C 180,E1 -1167.288,E2 -1167.288} C_VEL
LIN {X 0,Y 594.24,Z 557.2,A -85,B 0,C 180,E1 -1167.966,E2 -1167.966} C_VEL
LIN {X 0,Y 594.239,Z 558.784,A -85,B 0,C 180,E1 -1169.322,E2 -1169.322} C_VEL
LIN {X 0,Y 594.236,Z 559,A -85,B 0,C 180,E1 -1170,E2 -1170} C_VEL
LIN {X 0,Y 594.247,Z 558.185,A -85,B 0,C 180,E1 -1171.355,E2 -1171.355} C_VEL
LIN {X 0,Y 594.24,Z 557.202,A -85,B 0,C 180,E1 -1172.033,E2 -1172.033} C_VEL
LIN {X 0,Y 594.225,Z 555.811,A -85,B 0,C 180,E1 -1172.711,E2 -1172.711} C_VEL
LIN {X 0,Y 594.289,Z 552.897,A -85,B 0,C 180,E1 -1173.729,E2 -1173.729} C_VEL
LIN {X 0,Y 594.241,Z 548.951,A -85,B 0,C 180,E1 -1174.748,E2 -1174.748} C_VEL
LIN {X 0,Y 594.304,Z 542.88,A -85,B 0,C 180,E1 -1175.939,E2 -1175.939} C_VEL
LIN {X 0,Y 594.307,Z 536.239,A -85,B 0,C 180,E1 -1176.962,E2 -1176.962} C_VEL
LIN {X 0,Y 594.359,Z 527.993,A -85,B 0,C 180,E1 -1177.986,E2 -1177.986} C_VEL
LIN {X 0,Y 594.382,Z 519.542,A -85,B 0,C 180,E1 -1178.842,E2 -1178.842} C_VEL
LIN {X 0,Y 594.426,Z 509.1,A -85,B 0,C 180,E1 -1179.699,E2 -1179.699} C_VEL
LIN {X 0,Y 594.494,Z 498.766,A -85,B 0,C 180,E1 -1180.386,E2 -1180.386} C_VEL
LIN {X 0,Y 594.559,Z 487.705,A -85,B 0,C 180,E1 -1180.974,E2 -1180.974} C_VEL
LIN {X 0,Y 594.568,Z 475.716,A -85,B 0,C 180,E1 -1181.464,E2 -1181.464} C_VEL
LIN {X 0,Y 594.598,Z 462.369,A -85,B 0,C 180,E1 -1181.851,E2 -1181.851} C_VEL
LIN {X 0,Y 594.671,Z 449.117,A -85,B 0,C 180,E1 -1182.087,E2 -1182.087} C_VEL
LIN {X 0,Y 594.626,Z 347.961,A -85,B 0,C 180,E1 -1183.315,E2 -1183.315} C_VEL
LIN {X 0,Y 594.436,Z 346.442,A -85,B 0,C 180,E1 -1183.351,E2 -1183.351} C_VEL
LIN {X 0,Y 594.511,Z 325.334,A -85,B 0,C 180,E1 -1186.129,E2 -1186.129} C_VEL
LIN {X 0,Y 594.606,Z 304.735,A -85,B 0,C 180,E1 -1188.877,E2 -1188.877} C_VEL
LIN {X 0,Y 594.7,Z 286.554,A -85,B 0,C 180,E1 -1191.339,E2 -1191.339} C_VEL
LIN {X 0,Y 594.734,Z 273.48,A -85,B 0,C 180,E1 -1193.136,E2 -1193.136} C_VEL
LIN {X 0,Y 594.325,Z 271.453,A -85,B 0,C 180,E1 -1193.452,E2 -1193.452} C_VEL
LIN {X 0,Y 594.348,Z 271.451,A -85,B 0,C 180,E1 -1196.015,E2 -1196.015} C_VEL
LIN {X 0,Y 594.373,Z 271.443,A -85,B 0,C 180,E1 -1198.998,E2 -1198.998} C_VEL
LIN {X 0,Y 594.368,Z 271.443,A -85,B 0,C 180,E1 -1201.641,E2 -1201.641} C_VEL
LIN {X 0,Y 594.375,Z 271.448,A -85,B 0,C 180,E1 -1204.58,E2 -1204.58} C_VEL
LIN {X 0,Y 594.381,Z 271.44,A -85,B 0,C 180,E1 -1207.607,E2 -1207.607} C_VEL
LIN {X 0,Y 594.362,Z 271.45,A -85,B 0,C 180,E1 -1210.567,E2 -1210.567} C_VEL
LIN {X 0,Y 594.349,Z 271.444,A -85,B 0,C 180,E1 -1213.3,E2 -1213.3} C_VEL
LIN {X 0,Y 594.357,Z 271.448,A -85,B 0,C 180,E1 -1216.161,E2 -1216.161} C_VEL
LIN {X 0,Y 594.374,Z 271.442,A -85,B 0,C 180,E1 -1219.178,E2 -1219.178} C_VEL
LIN {X 0,Y 594.373,Z 271.444,A -85,B 0,C 180,E1 -1222.058,E2 -1222.058} C_VEL
LIN {X 0,Y 594.359,Z 271.451,A -85,B 0,C 180,E1 -1224.675,E2 -1224.675} C_VEL
LIN {X 0,Y 594.375,Z 271.443,A -85,B 0,C 180,E1 -1227.088,E2 -1227.088} C_VEL
LIN {X 0,Y 594.369,Z 271.441,A -85,B 0,C 180,E1 -1229.674,E2 -1229.674} C_VEL
LIN {X 0,Y 594.372,Z 271.45,A -85,B 0,C 180,E1 -1232.539,E2 -1232.539} C_VEL
LIN {X 0,Y 594.369,Z 271.449,A -85,B 0,C 180,E1 -1234.807,E2 -1234.807} C_VEL
LIN {X 0,Y 594.362,Z 271.444,A -85,B 0,C 180,E1 -1237.265,E2 -1237.265} C_VEL
LIN {X 0,Y 594.372,Z 271.441,A -85,B 0,C 180,E1 -1239.946,E2 -1239.946} C_VEL
LIN {X 0,Y 594.388,Z 271.449,A -85,B 0,C 180,E1 -1242.807,E2 -1242.807} C_VEL
LIN {X 0,Y 594.386,Z 271.439,A -85,B 0,C 180,E1 -1245.826,E2 -1245.826} C_VEL
LIN {X 0,Y 594.391,Z 271.442,A -85,B 0,C 180,E1 -1248.404,E2 -1248.404} C_VEL
LIN {X 0,Y 594.38,Z 271.445,A -85,B 0,C 180,E1 -1251.158,E2 -1251.158} C_VEL
LIN {X 0,Y 594.361,Z 271.442,A -85,B 0,C 180,E1 -1253.891,E2 -1253.891} C_VEL
LIN {X 0,Y 594.383,Z 271.445,A -85,B 0,C 180,E1 -1256.611,E2 -1256.611} C_VEL
LIN {X 0,Y 594.413,Z 271.44,A -85,B 0,C 180,E1 -1259.323,E2 -1259.323} C_VEL
LIN {X 0,Y 594.4,Z 271.437,A -85,B 0,C 180,E1 -1262.033,E2 -1262.033} C_VEL
LIN {X 0,Y 594.388,Z 271.446,A -85,B 0,C 180,E1 -1264.748,E2 -1264.748} C_VEL
LIN {X 0,Y 594.39,Z 271.442,A -85,B 0,C 180,E1 -1267.473,E2 -1267.473} C_VEL
LIN {X 0,Y 594.386,Z 271.439,A -85,B 0,C 180,E1 -1270.216,E2 -1270.216} C_VEL
LIN {X 0,Y 594.365,Z 271.451,A -85,B 0,C 180,E1 -1272.983,E2 -1272.983} C_VEL
LIN {X 0,Y 594.358,Z 271.449,A -85,B 0,C 180,E1 -1275.326,E2 -1275.326} C_VEL
LIN {X 0,Y 593.68,Z 271.529,A -85,B 0,C 180,E1 -1275.892,E2 -1275.892} C_VEL
LIN {X 0,Y 590.808,Z 271.891,A -85,B 0,C 180,E1 -1276.81,E2 -1276.81} C_VEL
LIN {X 0,Y 588.396,Z 272.189,A -85,B 0,C 180,E1 -1277.549,E2 -1277.549} C_VEL
LIN {X 0,Y 587.376,Z 272.312,A -85,B 0,C 180,E1 -1278.119,E2 -1278.119} C_VEL
LIN {X 0,Y 587.301,Z 272.322,A -85,B 0,C 180,E1 -1278.312,E2 -1278.312} C_VEL
LIN {X 0,Y 587.329,Z 272.327,A -85,B 0,C 180,E1 -1281.038,E2 -1281.038} C_VEL
LIN {X 0,Y 587.308,Z 272.33,A -85,B 0,C 180,E1 -1283.26,E2 -1283.26} C_VEL
LIN {X 0,Y 587.323,Z 272.324,A -85,B 0,C 180,E1 -1285.518,E2 -1285.518} C_VEL
LIN {X 0,Y 587.338,Z 272.319,A -85,B 0,C 180,E1 -1287.819,E2 -1287.819} C_VEL
LIN {X 0,Y 587.32,Z 272.32,A -85,B 0,C 180,E1 -1290.508,E2 -1290.508} C_VEL
LIN {X 0,Y 587.325,Z 272.327,A -85,B 0,C 180,E1 -1293.398,E2 -1293.398} C_VEL
LIN {X 0,Y 587.288,Z 272.325,A -85,B 0,C 180,E1 -1295.901,E2 -1295.901} C_VEL
LIN {X 0,Y 587.315,Z 272.32,A -85,B 0,C 180,E1 -1298.481,E2 -1298.481} C_VEL
LIN {X 0,Y 587.334,Z 272.325,A -85,B 0,C 180,E1 -1301.158,E2 -1301.158} C_VEL
LIN {X 0,Y 587.303,Z 272.323,A -85,B 0,C 180,E1 -1304.112,E2 -1304.112} C_VEL
LIN {X 0,Y 587.303,Z 272.326,A -85,B 0,C 180,E1 -1306.993,E2 -1306.993} C_VEL
LIN {X 0,Y 587.3,Z 272.325,A -85,B 0,C 180,E1 -1309.985,E2 -1309.985} C_VEL
LIN {X 0,Y 587.31,Z 272.321,A -85,B 0,C 180,E1 -1312.39,E2 -1312.39} C_VEL
LIN {X 0,Y 587.337,Z 272.326,A -85,B 0,C 180,E1 -1315.655,E2 -1315.655} C_VEL
LIN {X 0,Y 587.333,Z 272.319,A -85,B 0,C 180,E1 -1318.231,E2 -1318.231} C_VEL
LIN {X 0,Y 587.342,Z 272.319,A -85,B 0,C 180,E1 -1320.869,E2 -1320.869} C_VEL
LIN {X 0,Y 587.318,Z 272.423,A -85,B 0,C 180,E1 -1322.789,E2 -1322.789} C_VEL
LIN {X 0,Y 587.392,Z 283.732,A -85,B 0,C 180,E1 -1324.866,E2 -1324.866} C_VEL
LIN {X 0,Y 587.337,Z 298.647,A -85,B 0,C 180,E1 -1327.568,E2 -1327.568} C_VEL
LIN {X 0,Y 587.867,Z 303.885,A -85,B 0,C 180,E1 -1327.647,E2 -1327.647} C_VEL
LIN {X 0,Y 587.727,Z 404.953,A -85,B 0,C 180,E1 -1328.9,E2 -1328.9} C_VEL
LIN {X 0,Y 587.667,Z 418.195,A -85,B 0,C 180,E1 -1329.205,E2 -1329.205} C_VEL
LIN {X 0,Y 587.6,Z 431.397,A -85,B 0,C 180,E1 -1329.66,E2 -1329.66} C_VEL
LIN {X 0,Y 587.502,Z 443.791,A -85,B 0,C 180,E1 -1330.249,E2 -1330.249} C_VEL
LIN {X 0,Y 587.421,Z 455.074,A -85,B 0,C 180,E1 -1330.94,E2 -1330.94} C_VEL
LIN {X 0,Y 587.393,Z 466.058,A -85,B 0,C 180,E1 -1331.786,E2 -1331.786} C_VEL
LIN {X 0,Y 587.28,Z 476.243,A -85,B 0,C 180,E1 -1332.77,E2 -1332.77} C_VEL
LIN {X 0,Y 587.252,Z 483.792,A -85,B 0,C 180,E1 -1333.666,E2 -1333.666} C_VEL
LIN {X 0,Y 587.219,Z 491.123,A -85,B 0,C 180,E1 -1334.734,E2 -1334.734} C_VEL
LIN {X 0,Y 587.196,Z 496.956,A -85,B 0,C 180,E1 -1335.808,E2 -1335.808} C_VEL
LIN {X 0,Y 587.166,Z 501.42,A -85,B 0,C 180,E1 -1336.855,E2 -1336.855} C_VEL
LIN {X 0,Y 587.18,Z 503.788,A -85,B 0,C 180,E1 -1337.559,E2 -1337.559} C_VEL
LIN {X 0,Y 587.162,Z 505.707,A -85,B 0,C 180,E1 -1338.26,E2 -1338.26} C_VEL
LIN {X 0,Y 587.168,Z 507.156,A -85,B 0,C 180,E1 -1338.96,E2 -1338.96} C_VEL
LIN {X 0,Y 587.15,Z 508.781,A -85,B 0,C 180,E1 -1340.354,E2 -1340.354} C_VEL
LIN {X 0,Y 587.127,Z 509,A -85,B 0,C 180,E1 -1341.048,E2 -1341.048} C_VEL
LIN {X 0,Y 587.146,Z 508.165,A -85,B 0,C 180,E1 -1342.434,E2 -1342.434} C_VEL
LIN {X 0,Y 587.189,Z 506.579,A -85,B 0,C 180,E1 -1343.427,E2 -1343.427} C_VEL
LIN {X 0,Y 587.156,Z 502.797,A -85,B 0,C 180,E1 -1344.85,E2 -1344.85} C_VEL
LIN {X 0,Y 587.183,Z 498.818,A -85,B 0,C 180,E1 -1345.882,E2 -1345.882} C_VEL
LIN {X 0,Y 587.236,Z 492.708,A -85,B 0,C 180,E1 -1347.085,E2 -1347.085} C_VEL
LIN {X 0,Y 587.253,Z 486.07,A -85,B 0,C 180,E1 -1348.114,E2 -1348.114} C_VEL
LIN {X 0,Y 587.307,Z 477.857,A -85,B 0,C 180,E1 -1349.143,E2 -1349.143} C_VEL
LIN {X 0,Y 587.33,Z 469.469,A -85,B 0,C 180,E1 -1350,E2 -1350} C_VEL
LIN {X 0,Y 587.388,Z 459.156,A -85,B 0,C 180,E1 -1350.857,E2 -1350.857} C_VEL
LIN {X 0,Y 587.449,Z 447.587,A -85,B 0,C 180,E1 -1351.629,E2 -1351.629} C_VEL
LIN {X 0,Y 587.561,Z 436.041,A -85,B 0,C 180,E1 -1352.228,E2 -1352.228} C_VEL
LIN {X 0,Y 587.598,Z 424.162,A -85,B 0,C 180,E1 -1352.7,E2 -1352.7} C_VEL
LIN {X 0,Y 587.645,Z 411.279,A -85,B 0,C 180,E1 -1353.064,E2 -1353.064} C_VEL
LIN {X 0,Y 587.7,Z 399.076,A -85,B 0,C 180,E1 -1353.278,E2 -1353.278} C_VEL
LIN {X 0,Y 587.83,Z 301.69,A -85,B 0,C 180,E1 -1354.471,E2 -1354.471} C_VEL
LIN {X 0,Y 587.321,Z 298.629,A -85,B 0,C 180,E1 -1354.526,E2 -1354.526} C_VEL
LIN {X 0,Y 587.406,Z 283.768,A -85,B 0,C 180,E1 -1357.217,E2 -1357.217} C_VEL
LIN {X 0,Y 587.306,Z 272.329,A -85,B 0,C 180,E1 -1359.319,E2 -1359.319} C_VEL
LIN {X 0,Y 587.328,Z 272.327,A -85,B 0,C 180,E1 -1362.439,E2 -1362.439} C_VEL
LIN {X 0,Y 587.315,Z 272.321,A -85,B 0,C 180,E1 -1365.264,E2 -1365.264} C_VEL
LIN {X 0,Y 587.285,Z 272.324,A -85,B 0,C 180,E1 -1367.408,E2 -1367.408} C_VEL
LIN {X 0,Y 587.302,Z 272.322,A -85,B 0,C 180,E1 -1369.577,E2 -1369.577} C_VEL
LIN {X 0,Y 587.307,Z 272.321,A -85,B 0,C 180,E1 -1371.775,E2 -1371.775} C_VEL
LIN {X 0,Y 587.313,Z 272.326,A -85,B 0,C 180,E1 -1374.57,E2 -1374.57} C_VEL
LIN {X 0,Y 587.306,Z 272.329,A -85,B 0,C 180,E1 -1377.048,E2 -1377.048} C_VEL
LIN {X 0,Y 587.308,Z 272.324,A -85,B 0,C 180,E1 -1379.382,E2 -1379.382} C_VEL
LIN {X 0,Y 587.32,Z 272.319,A -85,B 0,C 180,E1 -1381.831,E2 -1381.831} C_VEL
LIN {X 0,Y 587.338,Z 272.318,A -85,B 0,C 180,E1 -1384.345,E2 -1384.345} C_VEL
LIN {X 0,Y 587.34,Z 272.32,A -85,B 0,C 180,E1 -1387.609,E2 -1387.609} C_VEL
LIN {X 0,Y 587.297,Z 272.322,A -85,B 0,C 180,E1 -1390.256,E2 -1390.256} C_VEL
LIN {X 0,Y 587.295,Z 272.331,A -85,B 0,C 180,E1 -1393.115,E2 -1393.115} C_VEL
LIN {X 0,Y 587.301,Z 272.322,A -85,B 0,C 180,E1 -1396.047,E2 -1396.047} C_VEL
LIN {X 0,Y 587.312,Z 272.323,A -85,B 0,C 180,E1 -1398.928,E2 -1398.928} C_VEL
LIN {X 0,Y 587.313,Z 272.33,A -85,B 0,C 180,E1 -1401.519,E2 -1401.519} C_VEL
LIN {X 0,Y 587.281,Z 272.326,A -85,B 0,C 180,E1 -1404.099,E2 -1404.099} C_VEL
LIN {X 0,Y 587.32,Z 272.319,A -85,B 0,C 180,E1 -1406.602,E2 -1406.602} C_VEL
LIN {X 0,Y 587.318,Z 272.321,A -85,B 0,C 180,E1 -1409.032,E2 -1409.032} C_VEL
LIN {X 0,Y 587.316,Z 272.326,A -85,B 0,C 180,E1 -1411.402,E2 -1411.402} C_VEL
LIN {X 0,Y 587.298,Z 272.331,A -85,B 0,C 180,E1 -1413.832,E2 -1413.832} C_VEL
LIN {X 0,Y 587.306,Z 272.321,A -85,B 0,C 180,E1 -1416.74,E2 -1416.74} C_VEL
LIN {X 0,Y 587.321,Z 272.327,A -85,B 0,C 180,E1 -1419.695,E2 -1419.695} C_VEL
LIN {X 0,Y 587.285,Z 272.335,A -85,B 0,C 180,E1 -1421.872,E2 -1421.872} C_VEL
LIN {X 0,Y 587.304,Z 272.322,A -85,B 0,C 180,E1 -1424.736,E2 -1424.736} C_VEL
LIN {X 0,Y 587.292,Z 272.323,A -85,B 0,C 180,E1 -1426.858,E2 -1426.858} C_VEL
LIN {X 0,Y 587.321,Z 272.323,A -85,B 0,C 180,E1 -1429.66,E2 -1429.66} C_VEL
LIN {X 0,Y 587.314,Z 272.325,A -85,B 0,C 180,E1 -1432.436,E2 -1432.436} C_VEL
LIN {X 0,Y 587.327,Z 272.318,A -85,B 0,C 180,E1 -1435.195,E2 -1435.195} C_VEL
LIN {X 0,Y 587.37,Z 272.319,A -85,B 0,C 180,E1 -1437.943,E2 -1437.943} C_VEL
LIN {X 0,Y 587.372,Z 272.317,A -85,B 0,C 180,E1 -1440.685,E2 -1440.685} C_VEL
LIN {X 0,Y 587.35,Z 272.32,A -85,B 0,C 180,E1 -1442.743,E2 -1442.743} C_VEL
LIN {X 0,Y 587.322,Z 272.319,A -85,B 0,C 180,E1 -1445.493,E2 -1445.493} C_VEL
LIN {X 0,Y 587.323,Z 272.326,A -85,B 0,C 180,E1 -1448.256,E2 -1448.256} C_VEL
LIN {X 0,Y 587.3,Z 272.324,A -85,B 0,C 180,E1 -1451.107,E2 -1451.107} C_VEL
LIN {X 0,Y 587.329,Z 272.319,A -85,B 0,C 180,E1 -1453.846,E2 -1453.846} C_VEL
LIN {X 0,Y 587.325,Z 272.327,A -85,B 0,C 180,E1 -1456.805,E2 -1456.805} C_VEL
LIN {X 0,Y 587.299,Z 272.322,A -85,B 0,C 180,E1 -1459.576,E2 -1459.576} C_VEL
LIN {X 0,Y 587.307,Z 272.321,A -85,B 0,C 180,E1 -1461.775,E2 -1461.775} C_VEL
LIN {X 0,Y 587.3,Z 272.332,A -85,B 0,C 180,E1 -1464.761,E2 -1464.761} C_VEL
LIN {X 0,Y 587.3,Z 272.322,A -85,B 0,C 180,E1 -1467.682,E2 -1467.682} C_VEL
LIN {X 0,Y 587.295,Z 272.323,A -85,B 0,C 180,E1 -1470.172,E2 -1470.172} C_VEL
LIN {X 0,Y 587.333,Z 272.327,A -85,B 0,C 180,E1 -1473.11,E2 -1473.11} C_VEL
LIN {X 0,Y 587.279,Z 272.324,A -85,B 0,C 180,E1 -1475.901,E2 -1475.901} C_VEL
LIN {X 0,Y 587.313,Z 272.321,A -85,B 0,C 180,E1 -1478.481,E2 -1478.481} C_VEL
LIN {X 0,Y 587.311,Z 272.331,A -85,B 0,C 180,E1 -1481.159,E2 -1481.159} C_VEL
LIN {X 0,Y 587.306,Z 272.321,A -85,B 0,C 180,E1 -1484.111,E2 -1484.111} C_VEL
LIN {X 0,Y 587.292,Z 272.328,A -85,B 0,C 180,E1 -1486.991,E2 -1486.991} C_VEL
LIN {X 0,Y 587.3,Z 272.326,A -85,B 0,C 180,E1 -1489.744,E2 -1489.744} C_VEL
LIN {X 0,Y 587.308,Z 272.321,A -85,B 0,C 180,E1 -1492.389,E2 -1492.389} C_VEL
LIN {X 0,Y 587.338,Z 272.325,A -85,B 0,C 180,E1 -1495.654,E2 -1495.654} C_VEL
LIN {X 0,Y 587.335,Z 272.318,A -85,B 0,C 180,E1 -1498.23,E2 -1498.23} C_VEL
LIN {X 0,Y 587.344,Z 272.317,A -85,B 0,C 180,E1 -1500.868,E2 -1500.868} C_VEL
LIN {X 0,Y 587.296,Z 272.332,A -85,B 0,C 180,E1 -1503.832,E2 -1503.832} C_VEL
LIN {X 0,Y 587.349,Z 272.476,A -85,B 0,C 180,E1 -1506.415,E2 -1506.415} C_VEL
LIN {X 0,Y 587.887,Z 276.493,A -85,B 0,C 180,E1 -1507.001,E2 -1507.001} C_VEL
LIN {X 0,Y 587.763,Z 296.076,A -85,B 0,C 180,E1 -1509.71,E2 -1509.71} C_VEL
LIN {X 0,Y 587.587,Z 316.02,A -85,B 0,C 180,E1 -1512.421,E2 -1512.421} C_VEL
LIN {X 0,Y 587.481,Z 337.294,A -85,B 0,C 180,E1 -1515.273,E2 -1515.273} C_VEL
LIN {X 0,Y 587.403,Z 346.435,A -85,B 0,C 180,E1 -1516.486,E2 -1516.486} C_VEL
LIN {X 0,Y 587.842,Z 350.684,A -85,B 0,C 180,E1 -1516.562,E2 -1516.562} C_VEL
LIN {X 0,Y 587.722,Z 454.923,A -85,B 0,C 180,E1 -1517.855,E2 -1517.855} C_VEL
LIN {X 0,Y 587.67,Z 468.204,A -85,B 0,C 180,E1 -1518.16,E2 -1518.16} C_VEL
LIN {X 0,Y 587.624,Z 480.639,A -85,B 0,C 180,E1 -1518.586,E2 -1518.586} C_VEL
LIN {X 0,Y 587.555,Z 492.623,A -85,B 0,C 180,E1 -1519.141,E2 -1519.141} C_VEL
LIN {X 0,Y 587.468,Z 504.195,A -85,B 0,C 180,E1 -1519.836,E2 -1519.836} C_VEL
LIN {X 0,Y 587.393,Z 514.593,A -85,B 0,C 180,E1 -1520.617,E2 -1520.617} C_VEL
LIN {X 0,Y 587.322,Z 523.108,A -85,B 0,C 180,E1 -1521.397,E2 -1521.397} C_VEL
LIN {X 0,Y 587.274,Z 530.957,A -85,B 0,C 180,E1 -1522.262,E2 -1522.262} C_VEL
LIN {X 0,Y 587.231,Z 537.466,A -85,B 0,C 180,E1 -1523.126,E2 -1523.126} C_VEL
LIN {X 0,Y 587.236,Z 543.864,A -85,B 0,C 180,E1 -1524.161,E2 -1524.161} C_VEL
LIN {X 0,Y 587.147,Z 548.948,A -85,B 0,C 180,E1 -1525.193,E2 -1525.193} C_VEL
LIN {X 0,Y 587.213,Z 552.894,A -85,B 0,C 180,E1 -1526.225,E2 -1526.225} C_VEL
LIN {X 0,Y 587.132,Z 555.807,A -85,B 0,C 180,E1 -1527.255,E2 -1527.255} C_VEL
LIN {X 0,Y 587.139,Z 557.199,A -85,B 0,C 180,E1 -1527.942,E2 -1527.942} C_VEL
LIN {X 0,Y 587.14,Z 558.784,A -85,B 0,C 180,E1 -1529.314,E2 -1529.314} C_VEL
LIN {X 0,Y 587.137,Z 559,A -85,B 0,C 180,E1 -1530,E2 -1530} C_VEL
LIN {X 0,Y 587.147,Z 558.186,A -85,B 0,C 180,E1 -1531.371,E2 -1531.371} C_VEL
LIN {X 0,Y 587.139,Z 557.202,A -85,B 0,C 180,E1 -1532.057,E2 -1532.057} C_VEL
LIN {X 0,Y 587.132,Z 555.811,A -85,B 0,C 180,E1 -1532.744,E2 -1532.744} C_VEL
LIN {X 0,Y 587.213,Z 552.897,A -85,B 0,C 180,E1 -1533.774,E2 -1533.774} C_VEL
LIN {X 0,Y 587.147,Z 548.951,A -85,B 0,C 180,E1 -1534.806,E2 -1534.806} C_VEL
LIN {X 0,Y 587.217,Z 542.88,A -85,B 0,C 180,E1 -1536.011,E2 -1536.011} C_VEL
LIN {X 0,Y 587.244,Z 536.24,A -85,B 0,C 180,E1 -1537.046,E2 -1537.046} C_VEL
LIN {X 0,Y 587.299,Z 527.994,A -85,B 0,C 180,E1 -1538.083,E2 -1538.083} C_VEL
LIN {X 0,Y 587.343,Z 519.543,A -85,B 0,C 180,E1 -1538.949,E2 -1538.949} C_VEL
LIN {X 0,Y 587.413,Z 509.102,A -85,B 0,C 180,E1 -1539.816,E2 -1539.816} C_VEL
LIN {X 0,Y 587.513,Z 498.764,A -85,B 0,C 180,E1 -1540.511,E2 -1540.511} C_VEL
LIN {X 0,Y 587.567,Z 486.988,A -85,B 0,C 180,E1 -1541.141,E2 -1541.141} C_VEL
LIN {X 0,Y 587.602,Z 474.61,A -85,B 0,C 180,E1 -1541.639,E2 -1541.639} C_VEL
LIN {X 0,Y 587.681,Z 461.454,A -85,B 0,C 180,E1 -1542.014,E2 -1542.014} C_VEL
LIN {X 0,Y 587.726,Z 449.117,A -85,B 0,C 180,E1 -1542.232,E2 -1542.232} C_VEL
LIN {X 0,Y 587.718,Z 348.642,A -85,B 0,C 180,E1 -1543.466,E2 -1543.466} C_VEL
LIN {X 0,Y 587.405,Z 346.276,A -85,B 0,C 180,E1 -1543.535,E2 -1543.535} C_VEL
LIN {X 0,Y 587.542,Z 325.334,A -85,B 0,C 180,E1 -1546.325,E2 -1546.325} C_VEL
LIN {X 0,Y 587.683,Z 304.537,A -85,B 0,C 180,E1 -1549.135,E2 -1549.135} C_VEL
LIN {X 0,Y 587.807,Z 285.446,A -85,B 0,C 180,E1 -1551.755,E2 -1551.755} C_VEL
LIN {X 0,Y 587.8,Z 274.809,A -85,B 0,C 180,E1 -1553.238,E2 -1553.238} C_VEL
LIN {X 0,Y 587.309,Z 272.329,A -85,B 0,C 180,E1 -1553.632,E2 -1553.632} C_VEL
LIN {X 0,Y 587.295,Z 272.334,A -85,B 0,C 180,E1 -1556.28,E2 -1556.28} C_VEL
LIN {X 0,Y 587.342,Z 272.319,A -85,B 0,C 180,E1 -1559.132,E2 -1559.132} C_VEL
LIN {X 0,Y 587.338,Z 272.321,A -85,B 0,C 180,E1 -1561.834,E2 -1561.834} C_VEL
LIN {X 0,Y 587.337,Z 272.329,A -85,B 0,C 180,E1 -1564.346,E2 -1564.346} C_VEL
LIN {X 0,Y 587.337,Z 272.318,A -85,B 0,C 180,E1 -1567.608,E2 -1567.608} C_VEL
LIN {X 0,Y 587.305,Z 272.329,A -85,B 0,C 180,E1 -1570.255,E2 -1570.255} C_VEL
LIN {X 0,Y 587.304,Z 272.323,A -85,B 0,C 180,E1 -1573.117,E2 -1573.117} C_VEL
LIN {X 0,Y 587.309,Z 272.325,A -85,B 0,C 180,E1 -1576.048,E2 -1576.048} C_VEL
LIN {X 0,Y 587.334,Z 272.321,A -85,B 0,C 180,E1 -1578.925,E2 -1578.925} C_VEL
LIN {X 0,Y 587.32,Z 272.319,A -85,B 0,C 180,E1 -1581.52,E2 -1581.52} C_VEL
LIN {X 0,Y 587.289,Z 272.327,A -85,B 0,C 180,E1 -1584.1,E2 -1584.1} C_VEL
LIN {X 0,Y 587.325,Z 272.33,A -85,B 0,C 180,E1 -1586.603,E2 -1586.603} C_VEL
LIN {X 0,Y 587.334,Z 272.321,A -85,B 0,C 180,E1 -1589.034,E2 -1589.034} C_VEL
LIN {X 0,Y 587.32,Z 272.32,A -85,B 0,C 180,E1 -1591.403,E2 -1591.403} C_VEL
LIN {X 0,Y 587.336,Z 272.318,A -85,B 0,C 180,E1 -1593.823,E2 -1593.823} C_VEL
LIN {X 0,Y 587.321,Z 272.32,A -85,B 0,C 180,E1 -1595.993,E2 -1595.993} C_VEL
LIN {X 0,Y 587.319,Z 272.323,A -85,B 0,C 180,E1 -1598.226,E2 -1598.226} C_VEL
LIN {X 0,Y 587.348,Z 272.32,A -85,B 0,C 180,E1 -1601.151,E2 -1601.151} C_VEL
LIN {X 0,Y 587.323,Z 272.319,A -85,B 0,C 180,E1 -1604.025,E2 -1604.025} C_VEL
LIN {X 0,Y 587.359,Z 272.316,A -85,B 0,C 180,E1 -1606.154,E2 -1606.154} C_VEL
LIN {X 0,Y 587.339,Z 272.325,A -85,B 0,C 180,E1 -1608.962,E2 -1608.962} C_VEL
LIN {X 0,Y 587.362,Z 272.314,A -85,B 0,C 180,E1 -1611.745,E2 -1611.745} C_VEL
LIN {X 0,Y 587.356,Z 272.32,A -85,B 0,C 180,E1 -1614.507,E2 -1614.507} C_VEL
LIN {X 0,Y 587.367,Z 272.318,A -85,B 0,C 180,E1 -1617.257,E2 -1617.257} C_VEL
LIN {X 0,Y 587.382,Z 272.311,A -85,B 0,C 180,E1 -1620,E2 -1620} C_VEL
LIN {X 0,Y 587.37,Z 272.32,A -85,B 0,C 180,E1 -1622.743,E2 -1622.743} C_VEL
LIN {X 0,Y 587.352,Z 272.318,A -85,B 0,C 180,E1 -1625.493,E2 -1625.493} C_VEL
LIN {X 0,Y 587.365,Z 272.314,A -85,B 0,C 180,E1 -1628.255,E2 -1628.255} C_VEL
LIN {X 0,Y 587.346,Z 272.325,A -85,B 0,C 180,E1 -1631.134,E2 -1631.134} C_VEL
LIN {X 0,Y 587.362,Z 272.314,A -85,B 0,C 180,E1 -1634.261,E2 -1634.261} C_VEL
LIN {X 0,Y 587.344,Z 272.322,A -85,B 0,C 180,E1 -1637.406,E2 -1637.406} C_VEL
LIN {X 0,Y 587.301,Z 272.322,A -85,B 0,C 180,E1 -1638.312,E2 -1638.312} C_VEL
LIN {X 0,Y 586.664,Z 272.409,A -85,B 0,C 180,E1 -1638.884,E2 -1638.884} C_VEL
LIN {X 0,Y 583.842,Z 272.766,A -85,B 0,C 180,E1 -1639.813,E2 -1639.813} C_VEL
LIN {X 0,Y 581.431,Z 273.068,A -85,B 0,C 180,E1 -1640.56,E2 -1640.56} C_VEL
LIN {X 0,Y 580.376,Z 273.195,A -85,B 0,C 180,E1 -1641.136,E2 -1641.136} C_VEL
LIN {X 0,Y 580.28,Z 273.204,A -85,B 0,C 180,E1 -1641.331,E2 -1641.331} C_VEL
LIN {X 0,Y 580.289,Z 273.196,A -85,B 0,C 180,E1 -1644.317,E2 -1644.317} C_VEL
LIN {X 0,Y 580.281,Z 273.203,A -85,B 0,C 180,E1 -1647.402,E2 -1647.402} C_VEL
LIN {X 0,Y 580.275,Z 273.199,A -85,B 0,C 180,E1 -1649.774,E2 -1649.774} C_VEL
LIN {X 0,Y 580.293,Z 273.194,A -85,B 0,C 180,E1 -1652.201,E2 -1652.201} C_VEL
LIN {X 0,Y 580.291,Z 273.197,A -85,B 0,C 180,E1 -1654.697,E2 -1654.697} C_VEL
LIN {X 0,Y 580.294,Z 273.205,A -85,B 0,C 180,E1 -1657.269,E2 -1657.269} C_VEL
LIN {X 0,Y 580.283,Z 273.196,A -85,B 0,C 180,E1 -1660.27,E2 -1660.27} C_VEL
LIN {X 0,Y 580.256,Z 273.201,A -85,B 0,C 180,E1 -1662.709,E2 -1662.709} C_VEL
LIN {X 0,Y 580.249,Z 273.207,A -85,B 0,C 180,E1 -1665.612,E2 -1665.612} C_VEL
LIN {X 0,Y 580.248,Z 273.201,A -85,B 0,C 180,E1 -1668.229,E2 -1668.229} C_VEL
LIN {X 0,Y 580.264,Z 273.202,A -85,B 0,C 180,E1 -1670.965,E2 -1670.965} C_VEL
LIN {X 0,Y 580.244,Z 273.21,A -85,B 0,C 180,E1 -1673.595,E2 -1673.595} C_VEL
LIN {X 0,Y 580.275,Z 273.199,A -85,B 0,C 180,E1 -1676.143,E2 -1676.143} C_VEL
LIN {X 0,Y 580.261,Z 273.2,A -85,B 0,C 180,E1 -1678.614,E2 -1678.614} C_VEL
LIN {X 0,Y 580.285,Z 273.2,A -85,B 0,C 180,E1 -1681.024,E2 -1681.024} C_VEL
LIN {X 0,Y 580.295,Z 273.285,A -85,B 0,C 180,E1 -1682.721,E2 -1682.721} C_VEL
LIN {X 0,Y 580.364,Z 282.02,A -85,B 0,C 180,E1 -1684.348,E2 -1684.348} C_VEL
LIN {X 0,Y 580.298,Z 297.535,A -85,B 0,C 180,E1 -1687.198,E2 -1687.198} C_VEL
LIN {X 0,Y 580.293,Z 298.645,A -85,B 0,C 180,E1 -1687.401,E2 -1687.401} C_VEL
LIN {X 0,Y 580.983,Z 303.852,A -85,B 0,C 180,E1 -1687.485,E2 -1687.485} C_VEL
LIN {X 0,Y 580.779,Z 405.36,A -85,B 0,C 180,E1 -1688.761,E2 -1688.761} C_VEL
LIN {X 0,Y 580.716,Z 418.962,A -85,B 0,C 180,E1 -1689.083,E2 -1689.083} C_VEL
LIN {X 0,Y 580.646,Z 431.941,A -85,B 0,C 180,E1 -1689.544,E2 -1689.544} C_VEL
LIN {X 0,Y 580.532,Z 443.364,A -85,B 0,C 180,E1 -1690.094,E2 -1690.094} C_VEL
LIN {X 0,Y 580.421,Z 455.063,A -85,B 0,C 180,E1 -1690.816,E2 -1690.816} C_VEL
LIN {X 0,Y 580.332,Z 465.784,A -85,B 0,C 180,E1 -1691.648,E2 -1691.648} C_VEL
LIN {X 0,Y 580.276,Z 475.2,A -85,B 0,C 180,E1 -1692.557,E2 -1692.557} C_VEL
LIN {X 0,Y 580.186,Z 482.908,A -85,B 0,C 180,E1 -1693.462,E2 -1693.462} C_VEL
LIN {X 0,Y 580.155,Z 490.425,A -85,B 0,C 180,E1 -1694.544,E2 -1694.544} C_VEL
LIN {X 0,Y 580.114,Z 496.951,A -85,B 0,C 180,E1 -1695.742,E2 -1695.742} C_VEL
LIN {X 0,Y 580.095,Z 502.289,A -85,B 0,C 180,E1 -1697.049,E2 -1697.049} C_VEL
LIN {X 0,Y 580.063,Z 505.424,A -85,B 0,C 180,E1 -1698.114,E2 -1698.114} C_VEL
LIN {X 0,Y 580.075,Z 507.141,A -85,B 0,C 180,E1 -1698.926,E2 -1698.926} C_VEL
LIN {X 0,Y 580.057,Z 508.707,A -85,B 0,C 180,E1 -1700.234,E2 -1700.234} C_VEL
LIN {X 0,Y 580.026,Z 508.982,A -85,B 0,C 180,E1 -1700.938,E2 -1700.938} C_VEL
LIN {X 0,Y 580.06,Z 508.851,A -85,B 0,C 180,E1 -1701.64,E2 -1701.64} C_VEL
LIN {X 0,Y 580.062,Z 507.339,A -85,B 0,C 180,E1 -1703.041,E2 -1703.041} C_VEL
LIN {X 0,Y 580.067,Z 505.99,A -85,B 0,C 180,E1 -1703.74,E2 -1703.74} C_VEL
LIN {X 0,Y 580.072,Z 503.137,A -85,B 0,C 180,E1 -1704.787,E2 -1704.787} C_VEL
LIN {X 0,Y 580.106,Z 499.268,A -85,B 0,C 180,E1 -1705.832,E2 -1705.832} C_VEL
LIN {X 0,Y 580.122,Z 494.285,A -85,B 0,C 180,E1 -1706.875,E2 -1706.875} C_VEL
LIN {X 0,Y 580.14,Z 488.047,A -85,B 0,C 180,E1 -1707.918,E2 -1707.918} C_VEL
LIN {X 0,Y 580.231,Z 480.263,A -85,B 0,C 180,E1 -1708.959,E2 -1708.959} C_VEL
LIN {X 0,Y 580.275,Z 470.604,A -85,B 0,C 180,E1 -1710,E2 -1710} C_VEL
LIN {X 0,Y 580.364,Z 460.603,A -85,B 0,C 180,E1 -1710.868,E2 -1710.868} C_VEL
LIN {X 0,Y 580.438,Z 449.357,A -85,B 0,C 180,E1 -1711.648,E2 -1711.648} C_VEL
LIN {X 0,Y 580.554,Z 438.338,A -85,B 0,C 180,E1 -1712.255,E2 -1712.255} C_VEL
LIN {X 0,Y 580.644,Z 426.087,A -85,B 0,C 180,E1 -1712.776,E2 -1712.776} C_VEL
LIN {X 0,Y 580.692,Z 413.107,A -85,B 0,C 180,E1 -1713.166,E2 -1713.166} C_VEL
LIN {X 0,Y 580.786,Z 400.584,A -85,B 0,C 180,E1 -1713.404,E2 -1713.404} C_VEL
LIN {X 0,Y 580.975,Z 302.774,A -85,B 0,C 180,E1 -1714.619,E2 -1714.619} C_VEL
LIN {X 0,Y 580.304,Z 298.643,A -85,B 0,C 180,E1 -1714.69,E2 -1714.69} C_VEL
LIN {X 0,Y 580.39,Z 282.488,A -85,B 0,C 180,E1 -1717.655,E2 -1717.655} C_VEL
LIN {X 0,Y 580.259,Z 273.204,A -85,B 0,C 180,E1 -1719.389,E2 -1719.389} C_VEL
LIN {X 0,Y 580.288,Z 273.197,A -85,B 0,C 180,E1 -1721.882,E2 -1721.882} C_VEL
LIN {X 0,Y 580.284,Z 273.205,A -85,B 0,C 180,E1 -1724.735,E2 -1724.735} C_VEL
LIN {X 0,Y 580.25,Z 273.2,A -85,B 0,C 180,E1 -1727.626,E2 -1727.626} C_VEL
LIN {X 0,Y 580.281,Z 273.196,A -85,B 0,C 180,E1 -1729.824,E2 -1729.824} C_VEL
LIN {X 0,Y 580.254,Z 273.2,A -85,B 0,C 180,E1 -1732.054,E2 -1732.054} C_VEL
LIN {X 0,Y 580.26,Z 273.207,A -85,B 0,C 180,E1 -1734.715,E2 -1734.715} C_VEL
LIN {X 0,Y 580.251,Z 273.203,A -85,B 0,C 180,E1 -1737.404,E2 -1737.404} C_VEL
LIN {X 0,Y 580.256,Z 273.199,A -85,B 0,C 180,E1 -1739.775,E2 -1739.775} C_VEL
LIN {X 0,Y 580.29,Z 273.195,A -85,B 0,C 180,E1 -1742.202,E2 -1742.202} C_VEL
LIN {X 0,Y 580.285,Z 273.2,A -85,B 0,C 180,E1 -1744.697,E2 -1744.697} C_VEL
LIN {X 0,Y 580.289,Z 273.204,A -85,B 0,C 180,E1 -1747.27,E2 -1747.27} C_VEL
LIN {X 0,Y 580.278,Z 273.196,A -85,B 0,C 180,E1 -1750.268,E2 -1750.268} C_VEL
LIN {X 0,Y 580.24,Z 273.21,A -85,B 0,C 180,E1 -1753.386,E2 -1753.386} C_VEL
LIN {X 0,Y 580.24,Z 273.201,A -85,B 0,C 180,E1 -1756.338,E2 -1756.338} C_VEL
LIN {X 0,Y 580.28,Z 273.203,A -85,B 0,C 180,E1 -1759.154,E2 -1759.154} C_VEL
LIN {X 0,Y 580.279,Z 273.199,A -85,B 0,C 180,E1 -1761.929,E2 -1761.929} C_VEL
LIN {X 0,Y 580.232,Z 273.202,A -85,B 0,C 180,E1 -1764.451,E2 -1764.451} C_VEL
LIN {X 0,Y 580.287,Z 273.197,A -85,B 0,C 180,E1 -1766.974,E2 -1766.974} C_VEL
LIN {X 0,Y 580.282,Z 273.203,A -85,B 0,C 180,E1 -1769.424,E2 -1769.424} C_VEL
LIN {X 0,Y 580.259,Z 273.202,A -85,B 0,C 180,E1 -1772.15,E2 -1772.15} C_VEL
LIN {X 0,Y 580.245,Z 273.201,A -85,B 0,C 180,E1 -1774.917,E2 -1774.917} C_VEL
LIN {X 0,Y 580.286,Z 273.197,A -85,B 0,C 180,E1 -1777.197,E2 -1777.197} C_VEL
LIN {X 0,Y 580.271,Z 273.201,A -85,B 0,C 180,E1 -1779.437,E2 -1779.437} C_VEL
LIN {X 0,Y 580.245,Z 273.207,A -85,B 0,C 180,E1 -1781.644,E2 -1781.644} C_VEL
LIN {X 0,Y 580.273,Z 273.199,A -85,B 0,C 180,E1 -1784.546,E2 -1784.546} C_VEL
LIN {X 0,Y 580.252,Z 273.201,A -85,B 0,C 180,E1 -1786.695,E2 -1786.695} C_VEL
LIN {X 0,Y 580.272,Z 273.198,A -85,B 0,C 180,E1 -1788.826,E2 -1788.826} C_VEL
LIN {X 0,Y 580.304,Z 273.196,A -85,B 0,C 180,E1 -1791.643,E2 -1791.643} C_VEL
LIN {X 0,Y 580.302,Z 273.199,A -85,B 0,C 180,E1 -1794.44,E2 -1794.44} C_VEL
LIN {X 0,Y 580.307,Z 273.193,A -85,B 0,C 180,E1 -1797.223,E2 -1797.223} C_VEL
LIN {X 0,Y 580.351,Z 273.193,A -85,B 0,C 180,E1 -1800,E2 -1800} C_VEL
LIN {X 0,Y 580.316,Z 273.195,A -85,B 0,C 180,E1 -1802.776,E2 -1802.776} C_VEL
LIN {X 0,Y 580.292,Z 273.195,A -85,B 0,C 180,E1 -1805.56,E2 -1805.56} C_VEL
LIN {X 0,Y 580.295,Z 273.203,A -85,B 0,C 180,E1 -1808.356,E2 -1808.356} C_VEL
LIN {X 0,Y 580.271,Z 273.199,A -85,B 0,C 180,E1 -1811.174,E2 -1811.174} C_VEL
LIN {X 0,Y 580.293,Z 273.196,A -85,B 0,C 180,E1 -1814.018,E2 -1814.018} C_VEL
LIN {X 0,Y 580.271,Z 273.204,A -85,B 0,C 180,E1 -1816.898,E2 -1816.898} C_VEL
LIN {X 0,Y 580.278,Z 273.196,A -85,B 0,C 180,E1 -1819.823,E2 -1819.823} C_VEL
LIN {X 0,Y 580.253,Z 273.2,A -85,B 0,C 180,E1 -1822.053,E2 -1822.053} C_VEL
LIN {X 0,Y 580.257,Z 273.208,A -85,B 0,C 180,E1 -1824.715,E2 -1824.715} C_VEL
LIN {X 0,Y 580.246,Z 273.203,A -85,B 0,C 180,E1 -1827.404,E2 -1827.404} C_VEL
LIN {X 0,Y 580.254,Z 273.2,A -85,B 0,C 180,E1 -1829.775,E2 -1829.775} C_VEL
LIN {X 0,Y 580.287,Z 273.196,A -85,B 0,C 180,E1 -1832.201,E2 -1832.201} C_VEL
LIN {X 0,Y 580.282,Z 273.201,A -85,B 0,C 180,E1 -1834.697,E2 -1834.697} C_VEL
LIN {X 0,Y 580.287,Z 273.203,A -85,B 0,C 180,E1 -1837.269,E2 -1837.269} C_VEL
LIN {X 0,Y 580.275,Z 273.197,A -85,B 0,C 180,E1 -1840.268,E2 -1840.268} C_VEL
LIN {X 0,Y 580.238,Z 273.21,A -85,B 0,C 180,E1 -1843.386,E2 -1843.386} C_VEL
LIN {X 0,Y 580.238,Z 273.201,A -85,B 0,C 180,E1 -1846.338,E2 -1846.338} C_VEL
LIN {X 0,Y 580.278,Z 273.203,A -85,B 0,C 180,E1 -1849.154,E2 -1849.154} C_VEL
LIN {X 0,Y 580.277,Z 273.199,A -85,B 0,C 180,E1 -1851.929,E2 -1851.929} C_VEL
LIN {X 0,Y 580.231,Z 273.202,A -85,B 0,C 180,E1 -1854.451,E2 -1854.451} C_VEL
LIN {X 0,Y 580.284,Z 273.198,A -85,B 0,C 180,E1 -1856.974,E2 -1856.974} C_VEL
LIN {X 0,Y 580.28,Z 273.204,A -85,B 0,C 180,E1 -1859.424,E2 -1859.424} C_VEL
LIN {X 0,Y 580.257,Z 273.203,A -85,B 0,C 180,E1 -1862.149,E2 -1862.149} C_VEL
LIN {X 0,Y 580.243,Z 273.203,A -85,B 0,C 180,E1 -1864.917,E2 -1864.917} C_VEL
LIN {X 0,Y 580.293,Z 273.311,A -85,B 0,C 180,E1 -1866.253,E2 -1866.253} C_VEL
LIN {X 0,Y 580.985,Z 278.19,A -85,B 0,C 180,E1 -1866.955,E2 -1866.955} C_VEL
LIN {X 0,Y 580.831,Z 297.406,A -85,B 0,C 180,E1 -1869.642,E2 -1869.642} C_VEL
LIN {X 0,Y 580.608,Z 317.35,A -85,B 0,C 180,E1 -1872.385,E2 -1872.385} C_VEL
LIN {X 0,Y 580.47,Z 338.624,A -85,B 0,C 180,E1 -1875.27,E2 -1875.27} C_VEL
LIN {X 0,Y 580.396,Z 346.518,A -85,B 0,C 180,E1 -1876.33,E2 -1876.33} C_VEL
LIN {X 0,Y 580.971,Z 352.472,A -85,B 0,C 180,E1 -1876.422,E2 -1876.422} C_VEL
LIN {X 0,Y 580.783,Z 454.923,A -85,B 0,C 180,E1 -1877.707,E2 -1877.707} C_VEL
LIN {X 0,Y 580.729,Z 468.204,A -85,B 0,C 180,E1 -1878.016,E2 -1878.016} C_VEL
LIN {X 0,Y 580.675,Z 480.362,A -85,B 0,C 180,E1 -1878.436,E2 -1878.436} C_VEL
LIN {X 0,Y 580.575,Z 492.621,A -85,B 0,C 180,E1 -1879.008,E2 -1879.008} C_VEL
LIN {X 0,Y 580.446,Z 504.196,A -85,B 0,C 180,E1 -1879.712,E2 -1879.712} C_VEL
LIN {X 0,Y 580.343,Z 514.594,A -85,B 0,C 180,E1 -1880.502,E2 -1880.502} C_VEL
LIN {X 0,Y 580.272,Z 523.108,A -85,B 0,C 180,E1 -1881.292,E2 -1881.292} C_VEL
LIN {X 0,Y 580.222,Z 530.957,A -85,B 0,C 180,E1 -1882.168,E2 -1882.168} C_VEL
LIN {X 0,Y 580.154,Z 538.647,A -85,B 0,C 180,E1 -1883.221,E2 -1883.221} C_VEL
LIN {X 0,Y 580.139,Z 545.678,A -85,B 0,C 180,E1 -1884.438,E2 -1884.438} C_VEL
LIN {X 0,Y 580.108,Z 550.37,A -85,B 0,C 180,E1 -1885.483,E2 -1885.483} C_VEL
LIN {X 0,Y 580.123,Z 553.956,A -85,B 0,C 180,E1 -1886.527,E2 -1886.527} C_VEL
LIN {X 0,Y 580.043,Z 555.807,A -85,B 0,C 180,E1 -1887.222,E2 -1887.222} C_VEL
LIN {X 0,Y 580.039,Z 557.198,A -85,B 0,C 180,E1 -1887.916,E2 -1887.916} C_VEL
LIN {X 0,Y 580.04,Z 558.784,A -85,B 0,C 180,E1 -1889.305,E2 -1889.305} C_VEL
LIN {X 0,Y 580.037,Z 559,A -85,B 0,C 180,E1 -1890,E2 -1890} C_VEL
LIN {X 0,Y 580.046,Z 558.186,A -85,B 0,C 180,E1 -1891.388,E2 -1891.388} C_VEL
LIN {X 0,Y 580.039,Z 557.201,A -85,B 0,C 180,E1 -1892.083,E2 -1892.083} C_VEL
LIN {X 0,Y 580.043,Z 555.811,A -85,B 0,C 180,E1 -1892.778,E2 -1892.778} C_VEL
LIN {X 0,Y 580.11,Z 552.897,A -85,B 0,C 180,E1 -1893.82,E2 -1893.82} C_VEL
LIN {X 0,Y 580.053,Z 548.951,A -85,B 0,C 180,E1 -1894.865,E2 -1894.865} C_VEL
LIN {X 0,Y 580.139,Z 542.88,A -85,B 0,C 180,E1 -1896.084,E2 -1896.084} C_VEL
LIN {X 0,Y 580.184,Z 536.241,A -85,B 0,C 180,E1 -1897.132,E2 -1897.132} C_VEL
LIN {X 0,Y 580.25,Z 527.994,A -85,B 0,C 180,E1 -1898.181,E2 -1898.181} C_VEL
LIN {X 0,Y 580.308,Z 519.543,A -85,B 0,C 180,E1 -1899.058,E2 -1899.058} C_VEL
LIN {X 0,Y 580.417,Z 509.103,A -85,B 0,C 180,E1 -1899.935,E2 -1899.935} C_VEL
LIN {X 0,Y 580.533,Z 498.763,A -85,B 0,C 180,E1 -1900.638,E2 -1900.638} C_VEL
LIN {X 0,Y 580.58,Z 487.417,A -85,B 0,C 180,E1 -1901.256,E2 -1901.256} C_VEL
LIN {X 0,Y 580.67,Z 475.78,A -85,B 0,C 180,E1 -1901.74,E2 -1901.74} C_VEL
LIN {X 0,Y 580.723,Z 463.281,A -85,B 0,C 180,E1 -1902.116,E2 -1902.116} C_VEL
LIN {X 0,Y 580.806,Z 450.632,A -85,B 0,C 180,E1 -1902.358,E2 -1902.358} C_VEL
LIN {X 0,Y 580.806,Z 349.315,A -85,B 0,C 180,E1 -1903.621,E2 -1903.621} C_VEL
LIN {X 0,Y 580.416,Z 346.442,A -85,B 0,C 180,E1 -1903.679,E2 -1903.679} C_VEL
LIN {X 0,Y 580.593,Z 324.005,A -85,B 0,C 180,E1 -1906.707,E2 -1906.707} C_VEL
LIN {X 0,Y 580.776,Z 302.582,A -85,B 0,C 180,E1 -1909.642,E2 -1909.642} C_VEL
LIN {X 0,Y 581.004,Z 281.457,A -85,B 0,C 180,E1 -1912.585,E2 -1912.585} C_VEL
LIN {X 0,Y 580.929,Z 276.441,A -85,B 0,C 180,E1 -1913.288,E2 -1913.288} C_VEL
LIN {X 0,Y 580.271,Z 273.207,A -85,B 0,C 180,E1 -1913.795,E2 -1913.795} C_VEL
LIN {X 0,Y 580.237,Z 273.208,A -85,B 0,C 180,E1 -1916.625,E2 -1916.625} C_VEL
LIN {X 0,Y 580.274,Z 273.199,A -85,B 0,C 180,E1 -1919.304,E2 -1919.304} C_VEL
LIN {X 0,Y 580.295,Z 273.205,A -85,B 0,C 180,E1 -1922.2,E2 -1922.2} C_VEL
LIN {X 0,Y 580.284,Z 273.202,A -85,B 0,C 180,E1 -1924.696,E2 -1924.696} C_VEL
LIN {X 0,Y 580.284,Z 273.196,A -85,B 0,C 180,E1 -1927.269,E2 -1927.269} C_VEL
LIN {X 0,Y 580.285,Z 273.204,A -85,B 0,C 180,E1 -1930.269,E2 -1930.269} C_VEL
LIN {X 0,Y 580.272,Z 273.204,A -85,B 0,C 180,E1 -1932.706,E2 -1932.706} C_VEL
LIN {X 0,Y 580.255,Z 273.2,A -85,B 0,C 180,E1 -1935.61,E2 -1935.61} C_VEL
LIN {X 0,Y 580.274,Z 273.203,A -85,B 0,C 180,E1 -1938.231,E2 -1938.231} C_VEL
LIN {X 0,Y 580.28,Z 273.2,A -85,B 0,C 180,E1 -1940.965,E2 -1940.965} C_VEL
LIN {X 0,Y 580.265,Z 273.198,A -85,B 0,C 180,E1 -1943.596,E2 -1943.596} C_VEL
LIN {X 0,Y 580.299,Z 273.197,A -85,B 0,C 180,E1 -1946.144,E2 -1946.144} C_VEL
LIN {X 0,Y 580.282,Z 273.206,A -85,B 0,C 180,E1 -1948.615,E2 -1948.615} C_VEL
LIN {X 0,Y 580.289,Z 273.199,A -85,B 0,C 180,E1 -1951.024,E2 -1951.024} C_VEL
LIN {X 0,Y 580.287,Z 273.195,A -85,B 0,C 180,E1 -1953.666,E2 -1953.666} C_VEL
LIN {X 0,Y 580.292,Z 273.194,A -85,B 0,C 180,E1 -1955.683,E2 -1955.683} C_VEL
LIN {X 0,Y 580.27,Z 273.198,A -85,B 0,C 180,E1 -1957.947,E2 -1957.947} C_VEL
LIN {X 0,Y 580.316,Z 273.199,A -85,B 0,C 180,E1 -1960.914,E2 -1960.914} C_VEL
LIN {X 0,Y 580.278,Z 273.196,A -85,B 0,C 180,E1 -1963.826,E2 -1963.826} C_VEL
LIN {X 0,Y 580.324,Z 273.191,A -85,B 0,C 180,E1 -1965.983,E2 -1965.983} C_VEL
LIN {X 0,Y 580.302,Z 273.204,A -85,B 0,C 180,E1 -1968.827,E2 -1968.827} C_VEL
LIN {X 0,Y 580.325,Z 273.191,A -85,B 0,C 180,E1 -1971.644,E2 -1971.644} C_VEL
LIN {X 0,Y 580.321,Z 273.195,A -85,B 0,C 180,E1 -1974.44,E2 -1974.44} C_VEL
LIN {X 0,Y 580.334,Z 273.195,A -85,B 0,C 180,E1 -1977.224,E2 -1977.224} C_VEL
LIN {X 0,Y 580.351,Z 273.187,A -85,B 0,C 180,E1 -1980,E2 -1980} C_VEL
LIN {X 0,Y 580.336,Z 273.197,A -85,B 0,C 180,E1 -1982.777,E2 -1982.777} C_VEL
LIN {X 0,Y 580.318,Z 273.193,A -85,B 0,C 180,E1 -1985.56,E2 -1985.56} C_VEL
LIN {X 0,Y 580.329,Z 273.191,A -85,B 0,C 180,E1 -1988.356,E2 -1988.356} C_VEL
LIN {X 0,Y 580.298,Z 273.202,A -85,B 0,C 180,E1 -1991.191,E2 -1991.191} C_VEL
LIN {X 0,Y 580.322,Z 273.191,A -85,B 0,C 180,E1 -1994.017,E2 -1994.017} C_VEL
LIN {X 0,Y 580.31,Z 273.2,A -85,B 0,C 180,E1 -1996.914,E2 -1996.914} C_VEL
LIN {X 0,Y 580.285,Z 273.197,A -85,B 0,C 180,E1 -1999.823,E2 -1999.823} C_VEL
LIN {X 0,Y 580.28,Z 273.204,A -85,B 0,C 180,E1 -2001.331,E2 -2001.331} C_VEL
LIN {X 0,Y 579.58,Z 273.286,A -85,B 0,C 180,E1 -2001.911,E2 -2001.911} C_VEL
LIN {X 0,Y 576.699,Z 273.648,A -85,B 0,C 180,E1 -2002.85,E2 -2002.85} C_VEL
LIN {X 0,Y 574.303,Z 273.944,A -85,B 0,C 180,E1 -2003.607,E2 -2003.607} C_VEL
LIN {X 0,Y 573.307,Z 274.065,A -85,B 0,C 180,E1 -2004.19,E2 -2004.19} C_VEL
LIN {X 0,Y 573.243,Z 274.074,A -85,B 0,C 180,E1 -2004.388,E2 -2004.388} C_VEL
LIN {X 0,Y 573.246,Z 274.079,A -85,B 0,C 180,E1 -2006.977,E2 -2006.977} C_VEL
LIN {X 0,Y 573.237,Z 274.08,A -85,B 0,C 180,E1 -2009.487,E2 -2009.487} C_VEL
LIN {X 0,Y 573.25,Z 274.073,A -85,B 0,C 180,E1 -2012.646,E2 -2012.646} C_VEL
LIN {X 0,Y 573.237,Z 274.083,A -85,B 0,C 180,E1 -2015.186,E2 -2015.186} C_VEL
LIN {X 0,Y 573.229,Z 274.077,A -85,B 0,C 180,E1 -2017.809,E2 -2017.809} C_VEL
LIN {X 0,Y 573.244,Z 274.073,A -85,B 0,C 180,E1 -2020.526,E2 -2020.526} C_VEL
LIN {X 0,Y 573.207,Z 274.083,A -85,B 0,C 180,E1 -2023.666,E2 -2023.666} C_VEL
LIN {X 0,Y 573.207,Z 274.079,A -85,B 0,C 180,E1 -2026.639,E2 -2026.639} C_VEL
LIN {X 0,Y 573.246,Z 274.083,A -85,B 0,C 180,E1 -2029.476,E2 -2029.476} C_VEL
LIN {X 0,Y 573.217,Z 274.078,A -85,B 0,C 180,E1 -2032.192,E2 -2032.192} C_VEL
LIN {X 0,Y 573.226,Z 274.081,A -85,B 0,C 180,E1 -2035.231,E2 -2035.231} C_VEL
LIN {X 0,Y 573.241,Z 274.081,A -85,B 0,C 180,E1 -2037.775,E2 -2037.775} C_VEL
LIN {X 0,Y 573.237,Z 274.076,A -85,B 0,C 180,E1 -2040.633,E2 -2040.633} C_VEL
LIN {X 0,Y 573.267,Z 274.167,A -85,B 0,C 180,E1 -2042.655,E2 -2042.655} C_VEL
LIN {X 0,Y 573.326,Z 282.382,A -85,B 0,C 180,E1 -2044.204,E2 -2044.204} C_VEL
LIN {X 0,Y 573.25,Z 297.903,A -85,B 0,C 180,E1 -2047.093,E2 -2047.093} C_VEL
LIN {X 0,Y 573.258,Z 298.644,A -85,B 0,C 180,E1 -2047.23,E2 -2047.23} C_VEL
LIN {X 0,Y 574.055,Z 303.754,A -85,B 0,C 180,E1 -2047.317,E2 -2047.317} C_VEL
LIN {X 0,Y 573.854,Z 405.405,A -85,B 0,C 180,E1 -2048.611,E2 -2048.611} C_VEL
LIN {X 0,Y 573.78,Z 418.874,A -85,B 0,C 180,E1 -2048.934,E2 -2048.934} C_VEL
LIN {X 0,Y 573.689,Z 431.362,A -85,B 0,C 180,E1 -2049.378,E2 -2049.378} C_VEL
LIN {X 0,Y 573.564,Z 442.937,A -85,B 0,C 180,E1 -2049.935,E2 -2049.935} C_VEL
LIN {X 0,Y 573.419,Z 455.072,A -85,B 0,C 180,E1 -2050.69,E2 -2050.69} C_VEL
LIN {X 0,Y 573.315,Z 465.512,A -85,B 0,C 180,E1 -2051.507,E2 -2051.507} C_VEL
LIN {X 0,Y 573.233,Z 474.135,A -85,B 0,C 180,E1 -2052.336,E2 -2052.336} C_VEL
LIN {X 0,Y 573.146,Z 482.44,A -85,B 0,C 180,E1 -2053.307,E2 -2053.307} C_VEL
LIN {X 0,Y 573.049,Z 489.695,A -85,B 0,C 180,E1 -2054.347,E2 -2054.347} C_VEL
LIN {X 0,Y 573.028,Z 495.746,A -85,B 0,C 180,E1 -2055.427,E2 -2055.427} C_VEL
LIN {X 0,Y 573.017,Z 500.582,A -85,B 0,C 180,E1 -2056.525,E2 -2056.525} C_VEL
LIN {X 0,Y 572.991,Z 504.19,A -85,B 0,C 180,E1 -2057.606,E2 -2057.606} C_VEL
LIN {X 0,Y 572.987,Z 507.122,A -85,B 0,C 180,E1 -2058.888,E2 -2058.888} C_VEL
LIN {X 0,Y 572.974,Z 508.631,A -85,B 0,C 180,E1 -2060.113,E2 -2060.113} C_VEL
LIN {X 0,Y 572.95,Z 508.896,A -85,B 0,C 180,E1 -2061.536,E2 -2061.536} C_VEL
LIN {X 0,Y 572.977,Z 508.412,A -85,B 0,C 180,E1 -2062.246,E2 -2062.246} C_VEL
LIN {X 0,Y 573.013,Z 506.652,A -85,B 0,C 180,E1 -2063.451,E2 -2063.451} C_VEL
LIN {X 0,Y 572.992,Z 503.472,A -85,B 0,C 180,E1 -2064.722,E2 -2064.722} C_VEL
LIN {X 0,Y 573.032,Z 499.715,A -85,B 0,C 180,E1 -2065.78,E2 -2065.78} C_VEL
LIN {X 0,Y 573.035,Z 494.855,A -85,B 0,C 180,E1 -2066.837,E2 -2066.837} C_VEL
LIN {X 0,Y 573.056,Z 488.751,A -85,B 0,C 180,E1 -2067.892,E2 -2067.892} C_VEL
LIN {X 0,Y 573.172,Z 481.18,A -85,B 0,C 180,E1 -2068.947,E2 -2068.947} C_VEL
LIN {X 0,Y 573.222,Z 471.716,A -85,B 0,C 180,E1 -2070,E2 -2070} C_VEL
LIN {X 0,Y 573.34,Z 461.98,A -85,B 0,C 180,E1 -2070.878,E2 -2070.878} C_VEL
LIN {X 0,Y 573.425,Z 451.116,A -85,B 0,C 180,E1 -2071.668,E2 -2071.668} C_VEL
LIN {X 0,Y 573.57,Z 438.79,A -85,B 0,C 180,E1 -2072.371,E2 -2072.371} C_VEL
LIN {X 0,Y 573.672,Z 426.71,A -85,B 0,C 180,E1 -2072.897,E2 -2072.897} C_VEL
LIN {X 0,Y 573.749,Z 414.032,A -85,B 0,C 180,E1 -2073.292,E2 -2073.292} C_VEL
LIN {X 0,Y 573.851,Z 400.634,A -85,B 0,C 180,E1 -2073.555,E2 -2073.555} C_VEL
LIN {X 0,Y 573.952,Z 302.987,A -85,B 0,C 180,E1 -2074.786,E2 -2074.786} C_VEL
LIN {X 0,Y 573.299,Z 298.537,A -85,B 0,C 180,E1 -2074.879,E2 -2074.879} C_VEL
LIN {X 0,Y 573.379,Z 283.101,A -85,B 0,C 180,E1 -2077.749,E2 -2077.749} C_VEL
LIN {X 0,Y 573.234,Z 274.153,A -85,B 0,C 180,E1 -2079.438,E2 -2079.438} C_VEL
LIN {X 0,Y 573.239,Z 274.077,A -85,B 0,C 180,E1 -2082.03,E2 -2082.03} C_VEL
LIN {X 0,Y 573.23,Z 274.08,A -85,B 0,C 180,E1 -2084.92,E2 -2084.92} C_VEL
LIN {X 0,Y 573.215,Z 274.076,A -85,B 0,C 180,E1 -2087.85,E2 -2087.85} C_VEL
LIN {X 0,Y 573.254,Z 274.082,A -85,B 0,C 180,E1 -2090.827,E2 -2090.827} C_VEL
LIN {X 0,Y 573.208,Z 274.077,A -85,B 0,C 180,E1 -2093.867,E2 -2093.867} C_VEL
LIN {X 0,Y 573.203,Z 274.082,A -85,B 0,C 180,E1 -2096.484,E2 -2096.484} C_VEL
LIN {X 0,Y 573.237,Z 274.078,A -85,B 0,C 180,E1 -2099.368,E2 -2099.368} C_VEL
LIN {X 0,Y 573.243,Z 274.073,A -85,B 0,C 180,E1 -2102.226,E2 -2102.226} C_VEL
LIN {X 0,Y 573.23,Z 274.08,A -85,B 0,C 180,E1 -2104.77,E2 -2104.77} C_VEL
LIN {X 0,Y 573.23,Z 274.076,A -85,B 0,C 180,E1 -2107.809,E2 -2107.809} C_VEL
LIN {X 0,Y 573.234,Z 274.075,A -85,B 0,C 180,E1 -2110.527,E2 -2110.527} C_VEL
LIN {X 0,Y 573.206,Z 274.087,A -85,B 0,C 180,E1 -2113.363,E2 -2113.363} C_VEL
LIN {X 0,Y 573.209,Z 274.077,A -85,B 0,C 180,E1 -2116.335,E2 -2116.335} C_VEL
LIN {X 0,Y 573.251,Z 274.082,A -85,B 0,C 180,E1 -2119.475,E2 -2119.475} C_VEL
LIN {X 0,Y 573.219,Z 274.077,A -85,B 0,C 180,E1 -2122.191,E2 -2122.191} C_VEL
LIN {X 0,Y 573.229,Z 274.08,A -85,B 0,C 180,E1 -2125.23,E2 -2125.23} C_VEL
LIN {X 0,Y 573.24,Z 274.075,A -85,B 0,C 180,E1 -2128.184,E2 -2128.184} C_VEL
LIN {X 0,Y 573.241,Z 274.073,A -85,B 0,C 180,E1 -2130.632,E2 -2130.632} C_VEL
LIN {X 0,Y 573.196,Z 274.086,A -85,B 0,C 180,E1 -2133.517,E2 -2133.517} C_VEL
LIN {X 0,Y 573.213,Z 274.081,A -85,B 0,C 180,E1 -2136.133,E2 -2136.133} C_VEL
LIN {X 0,Y 573.252,Z 274.073,A -85,B 0,C 180,E1 -2139.173,E2 -2139.173} C_VEL
LIN {X 0,Y 573.204,Z 274.081,A -85,B 0,C 180,E1 -2141.41,E2 -2141.41} C_VEL
LIN {X 0,Y 573.222,Z 274.081,A -85,B 0,C 180,E1 -2143.621,E2 -2143.621} C_VEL
LIN {X 0,Y 573.259,Z 274.078,A -85,B 0,C 180,E1 -2145.806,E2 -2145.806} C_VEL
LIN {X 0,Y 573.231,Z 274.075,A -85,B 0,C 180,E1 -2148.764,E2 -2148.764} C_VEL
LIN {X 0,Y 573.247,Z 274.074,A -85,B 0,C 180,E1 -2151.54,E2 -2151.54} C_VEL
LIN {X 0,Y 573.272,Z 274.076,A -85,B 0,C 180,E1 -2154.371,E2 -2154.371} C_VEL
LIN {X 0,Y 573.309,Z 274.069,A -85,B 0,C 180,E1 -2157.892,E2 -2157.892} C_VEL
LIN {X 0,Y 573.317,Z 274.068,A -85,B 0,C 180,E1 -2160.702,E2 -2160.702} C_VEL
LIN {X 0,Y 573.282,Z 274.071,A -85,B 0,C 180,E1 -2162.811,E2 -2162.811} C_VEL
LIN {X 0,Y 573.262,Z 274.071,A -85,B 0,C 180,E1 -2165.628,E2 -2165.628} C_VEL
LIN {X 0,Y 573.24,Z 274.084,A -85,B 0,C 180,E1 -2168.46,E2 -2168.46} C_VEL
LIN {X 0,Y 573.239,Z 274.074,A -85,B 0,C 180,E1 -2171.313,E2 -2171.313} C_VEL
LIN {X 0,Y 573.263,Z 274.078,A -85,B 0,C 180,E1 -2174.415,E2 -2174.415} C_VEL
LIN {X 0,Y 573.222,Z 274.079,A -85,B 0,C 180,E1 -2177.113,E2 -2177.113} C_VEL
LIN {X 0,Y 573.236,Z 274.075,A -85,B 0,C 180,E1 -2180.077,E2 -2180.077} C_VEL
LIN {X 0,Y 573.223,Z 274.079,A -85,B 0,C 180,E1 -2182.338,E2 -2182.338} C_VEL
LIN {X 0,Y 573.205,Z 274.08,A -85,B 0,C 180,E1 -2185.412,E2 -2185.412} C_VEL
LIN {X 0,Y 573.203,Z 274.082,A -85,B 0,C 180,E1 -2188.566,E2 -2188.566} C_VEL
LIN {X 0,Y 573.211,Z 274.087,A -85,B 0,C 180,E1 -2190.994,E2 -2190.994} C_VEL
LIN {X 0,Y 573.245,Z 274.075,A -85,B 0,C 180,E1 -2193.52,E2 -2193.52} C_VEL
LIN {X 0,Y 573.191,Z 274.079,A -85,B 0,C 180,E1 -2196.053,E2 -2196.053} C_VEL
LIN {X 0,Y 573.234,Z 274.077,A -85,B 0,C 180,E1 -2198.702,E2 -2198.702} C_VEL
LIN {X 0,Y 573.198,Z 274.082,A -85,B 0,C 180,E1 -2201.589,E2 -2201.589} C_VEL
LIN {X 0,Y 573.22,Z 274.076,A -85,B 0,C 180,E1 -2204.335,E2 -2204.335} C_VEL
LIN {X 0,Y 573.219,Z 274.086,A -85,B 0,C 180,E1 -2207.361,E2 -2207.361} C_VEL
LIN {X 0,Y 573.229,Z 274.074,A -85,B 0,C 180,E1 -2210.391,E2 -2210.391} C_VEL
LIN {X 0,Y 573.225,Z 274.079,A -85,B 0,C 180,E1 -2213.075,E2 -2213.075} C_VEL
LIN {X 0,Y 573.253,Z 274.079,A -85,B 0,C 180,E1 -2215.67,E2 -2215.67} C_VEL
LIN {X 0,Y 573.238,Z 274.075,A -85,B 0,C 180,E1 -2218.184,E2 -2218.184} C_VEL
LIN {X 0,Y 573.239,Z 274.074,A -85,B 0,C 180,E1 -2220.632,E2 -2220.632} C_VEL
LIN {X 0,Y 573.195,Z 274.088,A -85,B 0,C 180,E1 -2223.517,E2 -2223.517} C_VEL
LIN {X 0,Y 573.258,Z 274.183,A -85,B 0,C 180,E1 -2226.111,E2 -2226.111} C_VEL
LIN {X 0,Y 574.04,Z 279.834,A -85,B 0,C 180,E1 -2226.934,E2 -2226.934} C_VEL
LIN {X 0,Y 573.901,Z 298.736,A -85,B 0,C 180,E1 -2229.573,E2 -2229.573} C_VEL
LIN {X 0,Y 573.619,Z 318.813,A -85,B 0,C 180,E1 -2232.366,E2 -2232.366} C_VEL
LIN {X 0,Y 573.473,Z 339.763,A -85,B 0,C 180,E1 -2235.242,E2 -2235.242} C_VEL
LIN {X 0,Y 573.409,Z 346.518,A -85,B 0,C 180,E1 -2236.161,E2 -2236.161} C_VEL
LIN {X 0,Y 574.084,Z 352.472,A -85,B 0,C 180,E1 -2236.256,E2 -2236.256} C_VEL
LIN {X 0,Y 573.864,Z 454.923,A -85,B 0,C 180,E1 -2237.557,E2 -2237.557} C_VEL
LIN {X 0,Y 573.785,Z 468.203,A -85,B 0,C 180,E1 -2237.869,E2 -2237.869} C_VEL
LIN {X 0,Y 573.703,Z 480.364,A -85,B 0,C 180,E1 -2238.294,E2 -2238.294} C_VEL
LIN {X 0,Y 573.589,Z 492.634,A -85,B 0,C 180,E1 -2238.874,E2 -2238.874} C_VEL
LIN {X 0,Y 573.438,Z 504.194,A -85,B 0,C 180,E1 -2239.585,E2 -2239.585} C_VEL
LIN {X 0,Y 573.33,Z 514.596,A -85,B 0,C 180,E1 -2240.385,E2 -2240.385} C_VEL
LIN {X 0,Y 573.241,Z 523.108,A -85,B 0,C 180,E1 -2241.184,E2 -2241.184} C_VEL
LIN {X 0,Y 573.161,Z 530.957,A -85,B 0,C 180,E1 -2242.071,E2 -2242.071} C_VEL
LIN {X 0,Y 573.073,Z 538.951,A -85,B 0,C 180,E1 -2243.185,E2 -2243.185} C_VEL
LIN {X 0,Y 573.07,Z 545.678,A -85,B 0,C 180,E1 -2244.369,E2 -2244.369} C_VEL
LIN {X 0,Y 573.029,Z 550.37,A -85,B 0,C 180,E1 -2245.427,E2 -2245.427} C_VEL
LIN {X 0,Y 573.022,Z 553.956,A -85,B 0,C 180,E1 -2246.484,E2 -2246.484} C_VEL
LIN {X 0,Y 572.959,Z 555.807,A -85,B 0,C 180,E1 -2247.187,E2 -2247.187} C_VEL
LIN {X 0,Y 572.938,Z 557.197,A -85,B 0,C 180,E1 -2247.891,E2 -2247.891} C_VEL
LIN {X 0,Y 572.94,Z 558.785,A -85,B 0,C 180,E1 -2249.297,E2 -2249.297} C_VEL
LIN {X 0,Y 572.938,Z 559,A -85,B 0,C 180,E1 -2250,E2 -2250} C_VEL
LIN {X 0,Y 572.946,Z 558.187,A -85,B 0,C 180,E1 -2251.405,E2 -2251.405} C_VEL
LIN {X 0,Y 572.938,Z 557.2,A -85,B 0,C 180,E1 -2252.109,E2 -2252.109} C_VEL
LIN {X 0,Y 572.959,Z 555.811,A -85,B 0,C 180,E1 -2252.812,E2 -2252.812} C_VEL
LIN {X 0,Y 573.014,Z 552.897,A -85,B 0,C 180,E1 -2253.868,E2 -2253.868} C_VEL
LIN {X 0,Y 572.963,Z 548.951,A -85,B 0,C 180,E1 -2254.925,E2 -2254.925} C_VEL
LIN {X 0,Y 573.065,Z 542.879,A -85,B 0,C 180,E1 -2256.16,E2 -2256.16} C_VEL
